LIN {X 0.073,Y -402.750,Z 613.612,A 0.000,B 0.000,C 90.000,E1 146.087} C_DIS
LIN {X 0.112,Y -403.409,Z 613.600,A 0.000,B 0.000,C 90.000,E1 143.989} C_DIS
LIN {X -0.051,Y -403.995,Z 613.590,A 0.000,B 0.000,C 90.000,E1 142.271} C_DIS
LIN {X -0.134,Y -404.710,Z 613.579,A 0.000,B 0.000,C 90.000,E1 140.194} C_DIS
LIN {X 0.098,Y -405.120,Z 613.571,A 0.000,B 0.000,C 90.000,E1 138.771} C_DIS
LIN {X -0.008,Y -405.586,Z 613.560,A 0.000,B 0.000,C 90.000,E1 136.701} C_DIS
LIN {X -0.089,Y -405.878,Z 613.552,A 0.000,B 0.000,C 90.000,E1 135.324} C_DIS
LIN {X -0.078,Y -406.430,Z 613.538,A 0.000,B 0.000,C 90.000,E1 132.894} C_DIS
LIN {X 0.152,Y -406.905,Z 613.527,A 0.000,B 0.000,C 90.000,E1 130.782} C_DIS
LIN {X -0.174,Y -407.650,Z 613.515,A 0.000,B 0.000,C 90.000,E1 128.749} C_DIS
LIN {X 0.026,Y -415.541,Z 613.500,A 0.000,B 0.000,C 90.000,E1 125.964} C_DIS
LIN {X -0.040,Y -419.640,Z 613.490,A 0.000,B 0.000,C 90.000,E1 124.246} C_DIS
LIN {X -0.079,Y -419.686,Z 613.490,A 0.000,B 0.000,C 90.000,E1 124.246} C_DIS
LIN {X 0.070,Y -424.345,Z 613.489,A 0.000,B 0.000,C 90.000,E1 123.913} C_DIS
LIN {X -0.100,Y -446.604,Z 613.482,A 0.000,B 0.000,C 90.000,E1 122.752} C_DIS
LIN {X 0.090,Y -454.993,Z 613.479,A 0.000,B 0.000,C 90.000,E1 122.291} C_DIS
LIN {X -0.061,Y -463.376,Z 613.477,A 0.000,B 0.000,C 90.000,E1 121.848} C_DIS
LIN {X 0.207,Y -474.847,Z 613.473,A 0.000,B 0.000,C 90.000,E1 121.131} C_DIS
LIN {X -0.221,Y -484.333,Z 613.470,A 0.000,B 0.000,C 90.000,E1 120.590} C_DIS
LIN {X -0.006,Y -489.087,Z 613.468,A 0.000,B 0.000,C 90.000,E1 120.256} C_DIS
LIN {X 0.293,Y -495.307,Z 613.466,A 0.000,B 0.000,C 90.000,E1 119.795} C_DIS
LIN {X -0.178,Y -502.690,Z 613.463,A 0.000,B 0.000,C 90.000,E1 119.333} C_DIS
LIN {X 0.224,Y -507.199,Z 613.461,A 0.000,B 0.000,C 90.000,E1 118.949} C_DIS
LIN {X -0.050,Y -514.629,Z 613.458,A 0.000,B 0.000,C 90.000,E1 118.409} C_DIS
LIN {X 0.031,Y -521.564,Z 613.455,A 0.000,B 0.000,C 90.000,E1 117.847} C_DIS
LIN {X -0.121,Y -528.772,Z 613.451,A 0.000,B 0.000,C 90.000,E1 117.257} C_DIS
LIN {X -0.178,Y -535.593,Z 613.448,A 0.000,B 0.000,C 90.000,E1 116.668} C_DIS
LIN {X -0.109,Y -540.696,Z 613.445,A 0.000,B 0.000,C 90.000,E1 116.181} C_DIS
LIN {X -0.107,Y -545.705,Z 613.443,A 0.000,B 0.000,C 90.000,E1 115.668} C_DIS
LIN {X 0.123,Y -550.229,Z 613.440,A 0.000,B 0.000,C 90.000,E1 115.155} C_DIS
LIN {X 0.197,Y -554.784,Z 613.437,A 0.000,B 0.000,C 90.000,E1 114.591} C_DIS
LIN {X 0.157,Y -559.646,Z 613.433,A 0.000,B 0.000,C 90.000,E1 113.898} C_DIS
LIN {X 0.159,Y -563.793,Z 613.429,A 0.000,B 0.000,C 90.000,E1 113.206} C_DIS
LIN {X 0.098,Y -568.224,Z 613.424,A 0.000,B 0.000,C 90.000,E1 112.386} C_DIS
LIN {X -0.137,Y -572.184,Z 613.420,A 0.000,B 0.000,C 90.000,E1 111.589} C_DIS
LIN {X -0.247,Y -575.292,Z 613.416,A 0.000,B 0.000,C 90.000,E1 110.918} C_DIS
LIN {X 0.130,Y -578.678,Z 613.412,A 0.000,B 0.000,C 90.000,E1 110.066} C_DIS
LIN {X -0.162,Y -582.700,Z 613.406,A 0.000,B 0.000,C 90.000,E1 109.014} C_DIS
LIN {X -0.112,Y -584.647,Z 613.403,A 0.000,B 0.000,C 90.000,E1 108.471} C_DIS
LIN {X 0.181,Y -587.212,Z 613.398,A 0.000,B 0.000,C 90.000,E1 107.638} C_DIS
LIN {X 0.193,Y -590.315,Z 613.392,A 0.000,B 0.000,C 90.000,E1 106.567} C_DIS
LIN {X -0.158,Y -593.106,Z 613.386,A 0.000,B 0.000,C 90.000,E1 105.536} C_DIS
LIN {X -0.083,Y -600.448,Z 613.372,A 0.000,B 0.000,C 90.000,E1 102.883} C_DIS
LIN {X 0.280,Y -604.239,Z 613.364,A 0.000,B 0.000,C 90.000,E1 101.535} C_DIS
LIN {X 0.267,Y -607.275,Z 613.358,A 0.000,B 0.000,C 90.000,E1 100.489} C_DIS
LIN {X 0.040,Y -610.915,Z 613.351,A 0.000,B 0.000,C 90.000,E1 99.208} C_DIS
LIN {X -0.225,Y -614.306,Z 613.344,A 0.000,B 0.000,C 90.000,E1 97.936} C_DIS
LIN {X -0.105,Y -616.905,Z 613.338,A 0.000,B 0.000,C 90.000,E1 96.891} C_DIS
LIN {X -0.031,Y -619.305,Z 613.333,A 0.000,B 0.000,C 90.000,E1 95.853} C_DIS
LIN {X -0.293,Y -620.884,Z 613.328,A 0.000,B 0.000,C 90.000,E1 95.106} C_DIS
LIN {X 0.152,Y -623.278,Z 613.321,A 0.000,B 0.000,C 90.000,E1 93.784} C_DIS
LIN {X 0.261,Y -624.948,Z 613.315,A 0.000,B 0.000,C 90.000,E1 92.751} C_DIS
LIN {X -0.235,Y -626.386,Z 613.310,A 0.000,B 0.000,C 90.000,E1 91.776} C_DIS
LIN {X -0.174,Y -627.104,Z 613.307,A 0.000,B 0.000,C 90.000,E1 91.260} C_DIS
LIN {X -0.031,Y -628.115,Z 613.301,A 0.000,B 0.000,C 90.000,E1 90.229} C_DIS
LIN {X -0.229,Y -628.671,Z 613.297,A 0.000,B 0.000,C 90.000,E1 89.484} C_DIS
LIN {X 0.206,Y -628.976,Z 613.293,A 0.000,B 0.000,C 90.000,E1 88.682} C_DIS
LIN {X -0.240,Y -629.148,Z 613.287,A 0.000,B 0.000,C 90.000,E1 87.707} C_DIS
LIN {X 0.191,Y -629.030,Z 613.283,A 0.000,B 0.000,C 90.000,E1 86.906} C_DIS
LIN {X 0.137,Y -628.580,Z 613.276,A 0.000,B 0.000,C 90.000,E1 85.641} C_DIS
LIN {X 0.082,Y -627.646,Z 613.269,A 0.000,B 0.000,C 90.000,E1 84.375} C_DIS
LIN {X 0.007,Y -626.487,Z 613.262,A 0.000,B 0.000,C 90.000,E1 83.109} C_DIS
LIN {X 0.287,Y -625.243,Z 613.256,A 0.000,B 0.000,C 90.000,E1 82.064} C_DIS
LIN {X -0.152,Y -623.664,Z 613.250,A 0.000,B 0.000,C 90.000,E1 81.084} C_DIS
LIN {X 0.263,Y -620.907,Z 613.242,A 0.000,B 0.000,C 90.000,E1 79.511} C_DIS
LIN {X -0.139,Y -618.827,Z 613.236,A 0.000,B 0.000,C 90.000,E1 78.522} C_DIS
LIN {X 0.158,Y -616.553,Z 613.230,A 0.000,B 0.000,C 90.000,E1 77.465} C_DIS
LIN {X -0.174,Y -614.146,Z 613.225,A 0.000,B 0.000,C 90.000,E1 76.464} C_DIS
LIN {X 0.054,Y -611.588,Z 613.219,A 0.000,B 0.000,C 90.000,E1 75.408} C_DIS
LIN {X -0.192,Y -608.825,Z 613.213,A 0.000,B 0.000,C 90.000,E1 74.393} C_DIS
LIN {X 0.113,Y -605.900,Z 613.207,A 0.000,B 0.000,C 90.000,E1 73.323} C_DIS
LIN {X 0.065,Y -603.504,Z 613.203,A 0.000,B 0.000,C 90.000,E1 72.543} C_DIS
LIN {X -0.009,Y -600.882,Z 613.199,A 0.000,B 0.000,C 90.000,E1 71.764} C_DIS
LIN {X -0.211,Y -596.826,Z 613.193,A 0.000,B 0.000,C 90.000,E1 70.732} C_DIS
LIN {X -0.156,Y -593.507,Z 613.188,A 0.000,B 0.000,C 90.000,E1 69.934} C_DIS
LIN {X 0.153,Y -589.410,Z 613.183,A 0.000,B 0.000,C 90.000,E1 68.975} C_DIS
LIN {X 0.151,Y -585.015,Z 613.178,A 0.000,B 0.000,C 90.000,E1 68.050} C_DIS
LIN {X -0.175,Y -581.595,Z 613.174,A 0.000,B 0.000,C 90.000,E1 67.411} C_DIS
LIN {X -0.287,Y -577.056,Z 613.170,A 0.000,B 0.000,C 90.000,E1 66.613} C_DIS
LIN {X -0.138,Y -572.989,Z 613.166,A 0.000,B 0.000,C 90.000,E1 65.921} C_DIS
LIN {X 0.057,Y -569.490,Z 613.163,A 0.000,B 0.000,C 90.000,E1 65.357} C_DIS
LIN {X 0.042,Y -563.363,Z 613.159,A 0.000,B 0.000,C 90.000,E1 64.537} C_DIS
LIN {X -0.244,Y -560.182,Z 613.156,A 0.000,B 0.000,C 90.000,E1 64.152} C_DIS
LIN {X -0.145,Y -555.580,Z 613.153,A 0.000,B 0.000,C 90.000,E1 63.589} C_DIS
LIN {X -0.107,Y -549.415,Z 613.150,A 0.000,B 0.000,C 90.000,E1 62.948} C_DIS
LIN {X -0.330,Y -544.196,Z 613.147,A 0.000,B 0.000,C 90.000,E1 62.487} C_DIS
LIN {X -0.241,Y -539.657,Z 613.145,A 0.000,B 0.000,C 90.000,E1 62.103} C_DIS
LIN {X -0.278,Y -534.953,Z 613.143,A 0.000,B 0.000,C 90.000,E1 61.769} C_DIS
LIN {X 0.296,Y -528.777,Z 613.141,A 0.000,B 0.000,C 90.000,E1 61.307} C_DIS
LIN {X 0.186,Y -521.819,Z 613.139,A 0.000,B 0.000,C 90.000,E1 60.923} C_DIS
LIN {X 0.085,Y -516.888,Z 613.137,A 0.000,B 0.000,C 90.000,E1 60.667} C_DIS
LIN {X 0.102,Y -504.926,Z 613.134,A 0.000,B 0.000,C 90.000,E1 60.078} C_DIS
LIN {X 0.043,Y -486.360,Z 613.129,A 0.000,B 0.000,C 90.000,E1 59.203} C_DIS
LIN {X -0.144,Y -467.737,Z 613.124,A 0.000,B 0.000,C 90.000,E1 58.329} C_DIS
LIN {X -0.119,Y -449.331,Z 613.119,A 0.000,B 0.000,C 90.000,E1 57.375} C_DIS
LIN {X -0.171,Y -445.106,Z 613.118,A 0.000,B 0.000,C 90.000,E1 57.168} C_DIS
LIN {X 0.161,Y -445.092,Z 613.117,A 0.000,B 0.000,C 90.000,E1 57.120} C_DIS
LIN {X 0.186,Y -443.839,Z 613.114,A 0.000,B 0.000,C 90.000,E1 56.421} C_DIS
LIN {X 0.198,Y -434.691,Z 613.092,A 0.000,B 0.000,C 90.000,E1 52.477} C_DIS
LIN {X -0.024,Y -431.565,Z 613.083,A 0.000,B 0.000,C 90.000,E1 50.848} C_DIS
LIN {X -0.023,Y -429.048,Z 613.077,A 0.000,B 0.000,C 90.000,E1 49.828} C_DIS
LIN {X 0.098,Y -430.066,Z 613.068,A 0.000,B 0.000,C 90.000,E1 48.162} C_DIS
LIN {X -0.021,Y -431.027,Z 613.057,A 0.000,B 0.000,C 90.000,E1 46.176} C_DIS
LIN {X -0.117,Y -431.999,Z 613.045,A 0.000,B 0.000,C 90.000,E1 44.190} C_DIS
LIN {X -0.131,Y -432.905,Z 613.036,A 0.000,B 0.000,C 90.000,E1 42.528} C_DIS
LIN {X -0.096,Y -433.765,Z 613.027,A 0.000,B 0.000,C 90.000,E1 40.862} C_DIS
LIN {X 0.224,Y -434.710,Z 613.016,A 0.000,B 0.000,C 90.000,E1 38.830} C_DIS
LIN {X -0.256,Y -435.438,Z 613.007,A 0.000,B 0.000,C 90.000,E1 37.237} C_DIS
LIN {X -0.037,Y -435.880,Z 612.999,A 0.000,B 0.000,C 90.000,E1 35.884} C_DIS
LIN {X -0.132,Y -436.474,Z 612.988,A 0.000,B 0.000,C 90.000,E1 33.913} C_DIS
LIN {X -0.074,Y -437.035,Z 612.976,A 0.000,B 0.000,C 90.000,E1 31.592} C_DIS
LIN {X -0.113,Y -437.511,Z 612.964,A 0.000,B 0.000,C 90.000,E1 29.617} C_DIS
LIN {X -0.167,Y -437.939,Z 612.955,A 0.000,B 0.000,C 90.000,E1 27.975} C_DIS
LIN {X -0.031,Y -438.353,Z 612.946,A 0.000,B 0.000,C 90.000,E1 26.309} C_DIS
LIN {X 0.110,Y -438.845,Z 612.937,A 0.000,B 0.000,C 90.000,E1 24.643} C_DIS
LIN {X -0.092,Y -439.468,Z 612.926,A 0.000,B 0.000,C 90.000,E1 22.695} C_DIS
LIN {X -0.055,Y -440.105,Z 612.917,A 0.000,B 0.000,C 90.000,E1 21.046} C_DIS
LIN {X 0.004,Y -440.804,Z 612.908,A 0.000,B 0.000,C 90.000,E1 19.396} C_DIS
LIN {X 0.039,Y -441.756,Z 612.895,A 0.000,B 0.000,C 90.000,E1 17.094} C_DIS
LIN {X -0.007,Y -442.725,Z 612.884,A 0.000,B 0.000,C 90.000,E1 15.134} C_DIS
LIN {X -0.136,Y -444.216,Z 612.870,A 0.000,B 0.000,C 90.000,E1 12.535} C_DIS
LIN {X 0.020,Y -446.045,Z 612.855,A 0.000,B 0.000,C 90.000,E1 9.905} C_DIS
LIN {X 0.155,Y -447.600,Z 612.844,A 0.000,B 0.000,C 90.000,E1 7.936} C_DIS
LIN {X 0.013,Y -449.613,Z 612.832,A 0.000,B 0.000,C 90.000,E1 5.682} C_DIS
LIN {X -0.166,Y -451.886,Z 612.819,A 0.000,B 0.000,C 90.000,E1 3.440} C_DIS
LIN {X 0.140,Y -454.456,Z 612.807,A 0.000,B 0.000,C 90.000,E1 1.146} C_DIS
LIN {X 0.189,Y -458.356,Z 612.790,A 0.000,B 0.000,C 90.000,E1 358.167} C_DIS
LIN {X -0.013,Y -462.209,Z 612.776,A 0.000,B 0.000,C 90.000,E1 355.641} C_DIS
LIN {X -0.054,Y -465.357,Z 612.765,A 0.000,B 0.000,C 90.000,E1 353.742} C_DIS
LIN {X 0.026,Y -468.480,Z 612.755,A 0.000,B 0.000,C 90.000,E1 351.837} C_DIS
LIN {X -0.046,Y -470.984,Z 612.746,A 0.000,B 0.000,C 90.000,E1 350.274} C_DIS
LIN {X 0.063,Y -475.111,Z 612.732,A 0.000,B 0.000,C 90.000,E1 347.757} C_DIS
LIN {X -0.049,Y -479.579,Z 612.718,A 0.000,B 0.000,C 90.000,E1 345.283} C_DIS
LIN {X 0.220,Y -484.136,Z 612.705,A 0.000,B 0.000,C 90.000,E1 342.779} C_DIS
LIN {X -0.052,Y -487.075,Z 612.696,A 0.000,B 0.000,C 90.000,E1 341.275} C_DIS
LIN {X -0.085,Y -490.625,Z 612.686,A 0.000,B 0.000,C 90.000,E1 339.444} C_DIS
LIN {X -0.086,Y -493.494,Z 612.677,A 0.000,B 0.000,C 90.000,E1 337.922} C_DIS
LIN {X -0.120,Y -496.091,Z 612.669,A 0.000,B 0.000,C 90.000,E1 336.410} C_DIS
LIN {X -0.092,Y -498.501,Z 612.661,A 0.000,B 0.000,C 90.000,E1 334.897} C_DIS
LIN {X -0.027,Y -500.785,Z 612.652,A 0.000,B 0.000,C 90.000,E1 333.384} C_DIS
LIN {X -0.148,Y -502.972,Z 612.644,A 0.000,B 0.000,C 90.000,E1 331.897} C_DIS
LIN {X 0.014,Y -505.164,Z 612.635,A 0.000,B 0.000,C 90.000,E1 330.383} C_DIS
LIN {X -0.159,Y -507.817,Z 612.626,A 0.000,B 0.000,C 90.000,E1 328.614} C_DIS
LIN {X -0.131,Y -514.434,Z 612.606,A 0.000,B 0.000,C 90.000,E1 325.055} C_DIS
LIN {X 0.056,Y -519.892,Z 612.593,A 0.000,B 0.000,C 90.000,E1 322.683} C_DIS
LIN {X 0.002,Y -520.753,Z 612.591,A 0.000,B 0.000,C 90.000,E1 322.396} C_DIS
LIN {X -0.102,Y -522.945,Z 612.588,A 0.000,B 0.000,C 90.000,E1 321.823} C_DIS
LIN {X -0.148,Y -524.574,Z 612.586,A 0.000,B 0.000,C 90.000,E1 321.537} C_DIS
LIN {X -0.189,Y -525.990,Z 612.585,A 0.000,B 0.000,C 90.000,E1 321.251} C_DIS
LIN {X 0.048,Y -527.317,Z 612.584,A 0.000,B 0.000,C 90.000,E1 321.045} C_DIS
LIN {X -0.096,Y -531.585,Z 612.581,A 0.000,B 0.000,C 90.000,E1 320.642} C_DIS
LIN {X 0.056,Y -534.164,Z 612.580,A 0.000,B 0.000,C 90.000,E1 320.356} C_DIS
LIN {X -0.202,Y -538.452,Z 612.578,A 0.000,B 0.000,C 90.000,E1 319.989} C_DIS
LIN {X 0.201,Y -546.399,Z 612.574,A 0.000,B 0.000,C 90.000,E1 319.299} C_DIS
LIN {X -0.149,Y -553.775,Z 612.571,A 0.000,B 0.000,C 90.000,E1 318.771} C_DIS
LIN {X -0.073,Y -565.332,Z 612.566,A 0.000,B 0.000,C 90.000,E1 317.838} C_DIS
LIN {X 0.137,Y -582.769,Z 612.558,A 0.000,B 0.000,C 90.000,E1 316.458} C_DIS
LIN {X -0.011,Y -592.437,Z 612.554,A 0.000,B 0.000,C 90.000,E1 315.688} C_DIS
LIN {X -0.204,Y -600.545,Z 612.550,A 0.000,B 0.000,C 90.000,E1 315.000} C_DIS
LIN {X -0.188,Y -605.824,Z 612.547,A 0.000,B 0.000,C 90.000,E1 314.514} C_DIS
LIN {X 0.077,Y -610.557,Z 612.545,A 0.000,B 0.000,C 90.000,E1 314.028} C_DIS
LIN {X -0.197,Y -616.178,Z 612.541,A 0.000,B 0.000,C 90.000,E1 313.461} C_DIS
LIN {X 0.289,Y -621.962,Z 612.538,A 0.000,B 0.000,C 90.000,E1 312.771} C_DIS
LIN {X -0.178,Y -629.472,Z 612.533,A 0.000,B 0.000,C 90.000,E1 311.919} C_DIS
LIN {X -0.168,Y -637.595,Z 612.527,A 0.000,B 0.000,C 90.000,E1 310.906} C_DIS
LIN {X 0.012,Y -645.331,Z 612.522,A 0.000,B 0.000,C 90.000,E1 309.886} C_DIS
LIN {X -0.148,Y -648.943,Z 612.519,A 0.000,B 0.000,C 90.000,E1 309.402} C_DIS
LIN {X -0.169,Y -652.357,Z 612.516,A 0.000,B 0.000,C 90.000,E1 308.910} C_DIS
LIN {X -0.245,Y -656.969,Z 612.512,A 0.000,B 0.000,C 90.000,E1 308.177} C_DIS
LIN {X -0.281,Y -661.142,Z 612.508,A 0.000,B 0.000,C 90.000,E1 307.443} C_DIS
LIN {X 0.204,Y -664.308,Z 612.505,A 0.000,B 0.000,C 90.000,E1 306.790} C_DIS
LIN {X -0.164,Y -667.776,Z 612.500,A 0.000,B 0.000,C 90.000,E1 306.091} C_DIS
LIN {X -0.111,Y -670.868,Z 612.496,A 0.000,B 0.000,C 90.000,E1 305.358} C_DIS
LIN {X 0.131,Y -673.678,Z 612.492,A 0.000,B 0.000,C 90.000,E1 304.612} C_DIS
LIN {X 0.011,Y -677.229,Z 612.487,A 0.000,B 0.000,C 90.000,E1 303.658} C_DIS
LIN {X 0.310,Y -680.526,Z 612.482,A 0.000,B 0.000,C 90.000,E1 302.673} C_DIS
LIN {X -0.110,Y -684.530,Z 612.475,A 0.000,B 0.000,C 90.000,E1 301.514} C_DIS
LIN {X -0.237,Y -688.382,Z 612.468,A 0.000,B 0.000,C 90.000,E1 300.335} C_DIS
LIN {X 0.045,Y -692.081,Z 612.462,A 0.000,B 0.000,C 90.000,E1 299.127} C_DIS
LIN {X 0.076,Y -694.898,Z 612.457,A 0.000,B 0.000,C 90.000,E1 298.180} C_DIS
LIN {X 0.224,Y -696.862,Z 612.453,A 0.000,B 0.000,C 90.000,E1 297.462} C_DIS
LIN {X -0.238,Y -698.624,Z 612.449,A 0.000,B 0.000,C 90.000,E1 296.796} C_DIS
LIN {X 0.025,Y -699.176,Z 612.448,A 0.000,B 0.000,C 90.000,E1 296.539} C_DIS
LIN {X -0.377,Y -699.690,Z 612.445,A 0.000,B 0.000,C 90.000,E1 296.104} C_DIS
LIN {X -0.108,Y -699.900,Z 612.444,A 0.000,B 0.000,C 90.000,E1 295.848} C_DIS
LIN {X 0.161,Y -699.634,Z 612.442,A 0.000,B 0.000,C 90.000,E1 295.591} C_DIS
LIN {X -0.230,Y -698.669,Z 612.440,A 0.000,B 0.000,C 90.000,E1 295.155} C_DIS
LIN {X 0.037,Y -697.532,Z 612.438,A 0.000,B 0.000,C 90.000,E1 294.899} C_DIS
LIN {X -0.363,Y -694.083,Z 612.436,A 0.000,B 0.000,C 90.000,E1 294.463} C_DIS
LIN {X -0.236,Y -692.863,Z 612.435,A 0.000,B 0.000,C 90.000,E1 294.335} C_DIS
LIN {X -0.111,Y -690.927,Z 612.435,A 0.000,B 0.000,C 90.000,E1 294.207} C_DIS
LIN {X -0.313,Y -683.658,Z 612.433,A 0.000,B 0.000,C 90.000,E1 293.898} C_DIS
LIN {X -0.239,Y -681.111,Z 612.432,A 0.000,B 0.000,C 90.000,E1 293.823} C_DIS
LIN {X 0.181,Y -677.794,Z 612.432,A 0.000,B 0.000,C 90.000,E1 293.718} C_DIS
LIN {X -0.189,Y -675.746,Z 612.432,A 0.000,B 0.000,C 90.000,E1 293.695} C_DIS
LIN {X -0.053,Y -668.987,Z 612.431,A 0.000,B 0.000,C 90.000,E1 293.590} C_DIS
LIN {X 0.379,Y -647.864,Z 612.429,A 0.000,B 0.000,C 90.000,E1 293.259} C_DIS
LIN {X -0.161,Y -638.051,Z 612.428,A 0.000,B 0.000,C 90.000,E1 293.131} C_DIS
LIN {X 0.139,Y -628.502,Z 612.427,A 0.000,B 0.000,C 90.000,E1 292.898} C_DIS
LIN {X -0.291,Y -621.940,Z 612.426,A 0.000,B 0.000,C 90.000,E1 292.770} C_DIS
LIN {X -0.213,Y -605.336,Z 612.424,A 0.000,B 0.000,C 90.000,E1 292.280} C_DIS
LIN {X 0.108,Y -581.030,Z 612.419,A 0.000,B 0.000,C 90.000,E1 291.482} C_DIS
LIN {X -0.168,Y -565.314,Z 612.417,A 0.000,B 0.000,C 90.000,E1 291.046} C_DIS
LIN {X -0.257,Y -559.795,Z 612.415,A 0.000,B 0.000,C 90.000,E1 290.791} C_DIS
LIN {X 0.095,Y -558.001,Z 612.414,A 0.000,B 0.000,C 90.000,E1 290.556} C_DIS
LIN {X 0.052,Y -557.961,Z 612.414,A 0.000,B 0.000,C 90.000,E1 290.556} C_DIS
LIN {X 0.091,Y -557.398,Z 612.413,A 0.000,B 0.000,C 90.000,E1 290.301} C_DIS
LIN {X 0.150,Y -557.281,Z 612.407,A 0.000,B 0.000,C 90.000,E1 289.322} C_DIS
LIN {X -0.093,Y -557.311,Z 612.401,A 0.000,B 0.000,C 90.000,E1 288.236} C_DIS
LIN {X 0.195,Y -557.177,Z 612.395,A 0.000,B 0.000,C 90.000,E1 287.094} C_DIS
LIN {X 0.068,Y -556.689,Z 612.387,A 0.000,B 0.000,C 90.000,E1 285.717} C_DIS
LIN {X 0.190,Y -556.176,Z 612.381,A 0.000,B 0.000,C 90.000,E1 284.592} C_DIS
LIN {X 0.021,Y -555.336,Z 612.372,A 0.000,B 0.000,C 90.000,E1 282.939} C_DIS
LIN {X 0.124,Y -554.619,Z 612.364,A 0.000,B 0.000,C 90.000,E1 281.535} C_DIS
LIN {X -0.182,Y -553.624,Z 612.353,A 0.000,B 0.000,C 90.000,E1 279.613} C_DIS
LIN {X -0.170,Y -552.772,Z 612.344,A 0.000,B 0.000,C 90.000,E1 277.936} C_DIS
LIN {X -0.174,Y -552.018,Z 612.335,A 0.000,B 0.000,C 90.000,E1 276.258} C_DIS
LIN {X -0.209,Y -551.322,Z 612.324,A 0.000,B 0.000,C 90.000,E1 274.302} C_DIS
LIN {X 0.192,Y -550.796,Z 612.315,A 0.000,B 0.000,C 90.000,E1 272.579} C_DIS
LIN {X 0.001,Y -550.375,Z 612.305,A 0.000,B 0.000,C 90.000,E1 270.917} C_DIS
LIN {X -0.264,Y -549.900,Z 612.297,A 0.000,B 0.000,C 90.000,E1 269.542} C_DIS
LIN {X -0.045,Y -549.494,Z 612.291,A 0.000,B 0.000,C 90.000,E1 268.396} C_DIS
LIN {X -0.240,Y -548.822,Z 612.282,A 0.000,B 0.000,C 90.000,E1 266.731} C_DIS
LIN {X 0.022,Y -548.164,Z 612.274,A 0.000,B 0.000,C 90.000,E1 265.298} C_DIS
LIN {X 0.235,Y -547.667,Z 612.269,A 0.000,B 0.000,C 90.000,E1 264.432} C_DIS
LIN {X -0.037,Y -546.717,Z 612.261,A 0.000,B 0.000,C 90.000,E1 263.053} C_DIS
LIN {X 0.256,Y -545.757,Z 612.255,A 0.000,B 0.000,C 90.000,E1 261.894} C_DIS
LIN {X 0.174,Y -543.811,Z 612.244,A 0.000,B 0.000,C 90.000,E1 259.926} C_DIS
LIN {X 0.233,Y -541.938,Z 612.233,A 0.000,B 0.000,C 90.000,E1 257.937} C_DIS
LIN {X 0.293,Y -540.376,Z 612.224,A 0.000,B 0.000,C 90.000,E1 256.228} C_DIS
LIN {X 0.187,Y -539.313,Z 612.217,A 0.000,B 0.000,C 90.000,E1 255.102} C_DIS
LIN {X -0.187,Y -537.471,Z 612.208,A 0.000,B 0.000,C 90.000,E1 253.433} C_DIS
LIN {X 0.068,Y -535.761,Z 612.198,A 0.000,B 0.000,C 90.000,E1 251.692} C_DIS
LIN {X -0.163,Y -534.849,Z 612.194,A 0.000,B 0.000,C 90.000,E1 250.859} C_DIS
LIN {X -0.033,Y -533.391,Z 612.187,A 0.000,B 0.000,C 90.000,E1 249.699} C_DIS
LIN {X 0.075,Y -531.579,Z 612.181,A 0.000,B 0.000,C 90.000,E1 248.539} C_DIS
LIN {X -0.138,Y -529.662,Z 612.174,A 0.000,B 0.000,C 90.000,E1 247.411} C_DIS
LIN {X 0.114,Y -527.559,Z 612.168,A 0.000,B 0.000,C 90.000,E1 246.230} C_DIS
LIN {X 0.159,Y -525.906,Z 612.163,A 0.000,B 0.000,C 90.000,E1 245.357} C_DIS
LIN {X 0.093,Y -523.479,Z 612.157,A 0.000,B 0.000,C 90.000,E1 244.204} C_DIS
LIN {X 0.082,Y -521.617,Z 612.152,A 0.000,B 0.000,C 90.000,E1 243.332} C_DIS
LIN {X 0.192,Y -519.031,Z 612.145,A 0.000,B 0.000,C 90.000,E1 242.153} C_DIS
LIN {X -0.067,Y -515.600,Z 612.137,A 0.000,B 0.000,C 90.000,E1 240.717} C_DIS
LIN {X -0.138,Y -510.750,Z 612.126,A 0.000,B 0.000,C 90.000,E1 238.663} C_DIS
LIN {X 0.073,Y -507.787,Z 612.119,A 0.000,B 0.000,C 90.000,E1 237.454} C_DIS
LIN {X 0.121,Y -503.823,Z 612.111,A 0.000,B 0.000,C 90.000,E1 235.960} C_DIS
LIN {X -0.040,Y -499.741,Z 612.103,A 0.000,B 0.000,C 90.000,E1 234.482} C_DIS
LIN {X 0.164,Y -492.615,Z 612.088,A 0.000,B 0.000,C 90.000,E1 231.743} C_DIS
LIN {X -0.130,Y -489.510,Z 612.081,A 0.000,B 0.000,C 90.000,E1 230.561} C_DIS
LIN {X 0.007,Y -484.105,Z 612.069,A 0.000,B 0.000,C 90.000,E1 228.405} C_DIS
LIN {X 0.022,Y -480.295,Z 612.060,A 0.000,B 0.000,C 90.000,E1 226.863} C_DIS
LIN {X 0.169,Y -474.919,Z 612.048,A 0.000,B 0.000,C 90.000,E1 224.676} C_DIS
LIN {X -0.152,Y -469.932,Z 612.036,A 0.000,B 0.000,C 90.000,E1 222.528} C_DIS
LIN {X 0.021,Y -465.706,Z 612.026,A 0.000,B 0.000,C 90.000,E1 220.620} C_DIS
LIN {X -0.206,Y -461.640,Z 612.015,A 0.000,B 0.000,C 90.000,E1 218.749} C_DIS
LIN {X 0.187,Y -457.715,Z 612.005,A 0.000,B 0.000,C 90.000,E1 216.790} C_DIS
LIN {X -0.052,Y -453.977,Z 611.994,A 0.000,B 0.000,C 90.000,E1 214.898} C_DIS
LIN {X -0.086,Y -450.972,Z 611.985,A 0.000,B 0.000,C 90.000,E1 213.293} C_DIS
LIN {X 0.100,Y -446.838,Z 611.972,A 0.000,B 0.000,C 90.000,E1 211.003} C_DIS
LIN {X -0.057,Y -442.807,Z 611.960,A 0.000,B 0.000,C 90.000,E1 208.743} C_DIS
LIN {X -0.235,Y -439.885,Z 611.951,A 0.000,B 0.000,C 90.000,E1 207.129} C_DIS
LIN {X -0.077,Y -436.992,Z 611.941,A 0.000,B 0.000,C 90.000,E1 205.463} C_DIS
LIN {X 0.057,Y -433.568,Z 611.930,A 0.000,B 0.000,C 90.000,E1 203.462} C_DIS
LIN {X -0.081,Y -429.697,Z 611.917,A 0.000,B 0.000,C 90.000,E1 201.153} C_DIS
LIN {X -0.046,Y -426.363,Z 611.906,A 0.000,B 0.000,C 90.000,E1 199.141} C_DIS
LIN {X -0.166,Y -422.730,Z 611.893,A 0.000,B 0.000,C 90.000,E1 196.804} C_DIS
LIN {X -0.148,Y -419.886,Z 611.882,A 0.000,B 0.000,C 90.000,E1 194.773} C_DIS
LIN {X -0.116,Y -417.892,Z 611.874,A 0.000,B 0.000,C 90.000,E1 193.411} C_DIS
LIN {X 0.015,Y -414.241,Z 611.861,A 0.000,B 0.000,C 90.000,E1 191.007} C_DIS
LIN {X -0.112,Y -411.019,Z 611.848,A 0.000,B 0.000,C 90.000,E1 188.624} C_DIS
LIN {X -0.027,Y -408.734,Z 611.838,A 0.000,B 0.000,C 90.000,E1 186.891} C_DIS
LIN {X -0.063,Y -406.082,Z 611.827,A 0.000,B 0.000,C 90.000,E1 184.821} C_DIS
LIN {X 0.119,Y -402.200,Z 611.807,A 0.000,B 0.000,C 90.000,E1 181.318} C_DIS
LIN {X 0.189,Y -399.814,Z 611.792,A 0.000,B 0.000,C 90.000,E1 178.511} C_DIS
LIN {X -0.169,Y -398.107,Z 611.776,A 0.000,B 0.000,C 90.000,E1 175.755} C_DIS
LIN {X -0.179,Y -397.092,Z 611.759,A 0.000,B 0.000,C 90.000,E1 172.591} C_DIS
LIN {X 0.005,Y -396.606,Z 611.743,A 0.000,B 0.000,C 90.000,E1 169.746} C_DIS
LIN {X -0.087,Y -396.597,Z 611.731,A 0.000,B 0.000,C 90.000,E1 167.645} C_DIS
LIN {X 0.025,Y -397.009,Z 611.716,A 0.000,B 0.000,C 90.000,E1 164.810} C_DIS
LIN {X -0.162,Y -397.489,Z 611.704,A 0.000,B 0.000,C 90.000,E1 162.725} C_DIS
LIN {X -0.098,Y -398.006,Z 611.692,A 0.000,B 0.000,C 90.000,E1 160.604} C_DIS
LIN {X -0.101,Y -398.587,Z 611.682,A 0.000,B 0.000,C 90.000,E1 158.847} C_DIS
LIN {X -0.106,Y -399.318,Z 611.671,A 0.000,B 0.000,C 90.000,E1 156.741} C_DIS
LIN {X -0.065,Y -400.275,Z 611.657,A 0.000,B 0.000,C 90.000,E1 154.280} C_DIS
LIN {X -0.006,Y -400.776,Z 611.649,A 0.000,B 0.000,C 90.000,E1 152.871} C_DIS
LIN {X 0.056,Y -401.335,Z 611.642,A 0.000,B 0.000,C 90.000,E1 151.463} C_DIS
LIN {X 0.190,Y -402.117,Z 611.628,A 0.000,B 0.000,C 90.000,E1 148.997} C_DIS
LIN {X 0.110,Y -402.732,Z 611.616,A 0.000,B 0.000,C 90.000,E1 146.914} C_DIS
LIN {X 0.041,Y -403.487,Z 611.603,A 0.000,B 0.000,C 90.000,E1 144.482} C_DIS
LIN {X 0.012,Y -404.158,Z 611.591,A 0.000,B 0.000,C 90.000,E1 142.396} C_DIS
LIN {X -0.184,Y -404.951,Z 611.578,A 0.000,B 0.000,C 90.000,E1 139.989} C_DIS
LIN {X -0.087,Y -405.262,Z 611.572,A 0.000,B 0.000,C 90.000,E1 138.933} C_DIS
LIN {X 0.086,Y -405.723,Z 611.560,A 0.000,B 0.000,C 90.000,E1 136.824} C_DIS
LIN {X 0.018,Y -406.008,Z 611.553,A 0.000,B 0.000,C 90.000,E1 135.445} C_DIS
LIN {X 0.041,Y -406.507,Z 611.539,A 0.000,B 0.000,C 90.000,E1 133.014} C_DIS
LIN {X -0.188,Y -407.039,Z 611.526,A 0.000,B 0.000,C 90.000,E1 130.620} C_DIS
LIN {X 0.142,Y -407.689,Z 611.515,A 0.000,B 0.000,C 90.000,E1 128.669} C_DIS
LIN {X 0.092,Y -415.124,Z 611.501,A 0.000,B 0.000,C 90.000,E1 126.091} C_DIS
LIN {X 0.024,Y -416.038,Z 611.499,A 0.000,B 0.000,C 90.000,E1 125.758} C_DIS
LIN {X -0.191,Y -420.329,Z 611.489,A 0.000,B 0.000,C 90.000,E1 123.992} C_DIS
LIN {X -0.230,Y -420.357,Z 611.489,A 0.000,B 0.000,C 90.000,E1 123.992} C_DIS
LIN {X 0.079,Y -423.950,Z 611.487,A 0.000,B 0.000,C 90.000,E1 123.706} C_DIS
LIN {X 0.094,Y -431.463,Z 611.485,A 0.000,B 0.000,C 90.000,E1 123.293} C_DIS
LIN {X -0.141,Y -452.062,Z 611.479,A 0.000,B 0.000,C 90.000,E1 122.260} C_DIS
LIN {X 0.123,Y -458.727,Z 611.477,A 0.000,B 0.000,C 90.000,E1 121.878} C_DIS
LIN {X -0.150,Y -465.286,Z 611.475,A 0.000,B 0.000,C 90.000,E1 121.544} C_DIS
LIN {X -0.017,Y -476.739,Z 611.471,A 0.000,B 0.000,C 90.000,E1 120.846} C_DIS
LIN {X 0.137,Y -481.487,Z 611.470,A 0.000,B 0.000,C 90.000,E1 120.541} C_DIS
LIN {X -0.005,Y -489.375,Z 611.467,A 0.000,B 0.000,C 90.000,E1 120.050} C_DIS
LIN {X -0.010,Y -498.896,Z 611.463,A 0.000,B 0.000,C 90.000,E1 119.411} C_DIS
LIN {X 0.058,Y -503.560,Z 611.462,A 0.000,B 0.000,C 90.000,E1 119.077} C_DIS
LIN {X 0.152,Y -515.545,Z 611.457,A 0.000,B 0.000,C 90.000,E1 118.153} C_DIS
LIN {X -0.245,Y -520.061,Z 611.455,A 0.000,B 0.000,C 90.000,E1 117.847} C_DIS
LIN {X -0.199,Y -530.187,Z 611.450,A 0.000,B 0.000,C 90.000,E1 117.001} C_DIS
LIN {X -0.006,Y -535.818,Z 611.447,A 0.000,B 0.000,C 90.000,E1 116.488} C_DIS
LIN {X 0.002,Y -539.978,Z 611.445,A 0.000,B 0.000,C 90.000,E1 116.104} C_DIS
LIN {X -0.188,Y -546.468,Z 611.441,A 0.000,B 0.000,C 90.000,E1 115.463} C_DIS
LIN {X 0.136,Y -549.085,Z 611.440,A 0.000,B 0.000,C 90.000,E1 115.155} C_DIS
LIN {X 0.200,Y -553.345,Z 611.437,A 0.000,B 0.000,C 90.000,E1 114.643} C_DIS
LIN {X 0.353,Y -555.277,Z 611.436,A 0.000,B 0.000,C 90.000,E1 114.387} C_DIS
LIN {X -0.319,Y -559.305,Z 611.433,A 0.000,B 0.000,C 90.000,E1 113.898} C_DIS
LIN {X 0.018,Y -563.406,Z 611.429,A 0.000,B 0.000,C 90.000,E1 113.206} C_DIS
LIN {X -0.046,Y -567.962,Z 611.424,A 0.000,B 0.000,C 90.000,E1 112.386} C_DIS
LIN {X 0.247,Y -572.032,Z 611.420,A 0.000,B 0.000,C 90.000,E1 111.535} C_DIS
LIN {X 0.140,Y -575.213,Z 611.416,A 0.000,B 0.000,C 90.000,E1 110.865} C_DIS
LIN {X -0.020,Y -578.685,Z 611.411,A 0.000,B 0.000,C 90.000,E1 110.066} C_DIS
LIN {X 0.239,Y -582.782,Z 611.406,A 0.000,B 0.000,C 90.000,E1 108.960} C_DIS
LIN {X 0.293,Y -584.751,Z 611.403,A 0.000,B 0.000,C 90.000,E1 108.417} C_DIS
LIN {X -0.196,Y -586.585,Z 611.400,A 0.000,B 0.000,C 90.000,E1 107.928} C_DIS
LIN {X 0.045,Y -590.577,Z 611.392,A 0.000,B 0.000,C 90.000,E1 106.567} C_DIS
LIN {X 0.269,Y -593.422,Z 611.386,A 0.000,B 0.000,C 90.000,E1 105.481} C_DIS
LIN {X -0.218,Y -600.826,Z 611.372,A 0.000,B 0.000,C 90.000,E1 102.883} C_DIS
LIN {X 0.152,Y -604.672,Z 611.364,A 0.000,B 0.000,C 90.000,E1 101.535} C_DIS
LIN {X 0.144,Y -607.746,Z 611.358,A 0.000,B 0.000,C 90.000,E1 100.489} C_DIS
LIN {X -0.075,Y -611.430,Z 611.351,A 0.000,B 0.000,C 90.000,E1 99.208} C_DIS
LIN {X 0.010,Y -614.216,Z 611.345,A 0.000,B 0.000,C 90.000,E1 98.163} C_DIS
LIN {X -0.204,Y -617.511,Z 611.338,A 0.000,B 0.000,C 90.000,E1 96.891} C_DIS
LIN {X -0.122,Y -619.963,Z 611.333,A 0.000,B 0.000,C 90.000,E1 95.853} C_DIS
LIN {X 0.241,Y -621.548,Z 611.328,A 0.000,B 0.000,C 90.000,E1 95.049} C_DIS
LIN {X -0.246,Y -623.534,Z 611.323,A 0.000,B 0.000,C 90.000,E1 94.069} C_DIS
LIN {X -0.138,Y -625.275,Z 611.317,A 0.000,B 0.000,C 90.000,E1 93.037} C_DIS
LIN {X -0.029,Y -626.791,Z 611.311,A 0.000,B 0.000,C 90.000,E1 92.007} C_DIS
LIN {X 0.126,Y -628.111,Z 611.306,A 0.000,B 0.000,C 90.000,E1 90.974} C_DIS
LIN {X 0.283,Y -629.073,Z 611.300,A 0.000,B 0.000,C 90.000,E1 89.943} C_DIS
LIN {X -0.177,Y -629.667,Z 611.294,A 0.000,B 0.000,C 90.000,E1 88.969} C_DIS
LIN {X 0.015,Y -629.872,Z 611.289,A 0.000,B 0.000,C 90.000,E1 87.936} C_DIS
LIN {X 0.184,Y -629.777,Z 611.283,A 0.000,B 0.000,C 90.000,E1 86.906} C_DIS
LIN {X -0.209,Y -629.364,Z 611.277,A 0.000,B 0.000,C 90.000,E1 85.927} C_DIS
LIN {X 0.262,Y -628.912,Z 611.273,A 0.000,B 0.000,C 90.000,E1 85.122} C_DIS
LIN {X -0.188,Y -628.086,Z 611.267,A 0.000,B 0.000,C 90.000,E1 84.147} C_DIS
LIN {X 0.327,Y -627.412,Z 611.263,A 0.000,B 0.000,C 90.000,E1 83.337} C_DIS
LIN {X 0.323,Y -625.832,Z 611.256,A 0.000,B 0.000,C 90.000,E1 82.064} C_DIS
LIN {X -0.109,Y -624.223,Z 611.250,A 0.000,B 0.000,C 90.000,E1 81.084} C_DIS
LIN {X -0.075,Y -621.901,Z 611.243,A 0.000,B 0.000,C 90.000,E1 79.803} C_DIS
LIN {X 0.145,Y -619.834,Z 611.238,A 0.000,B 0.000,C 90.000,E1 78.757} C_DIS
LIN {X -0.150,Y -617.590,Z 611.232,A 0.000,B 0.000,C 90.000,E1 77.757} C_DIS
LIN {X -0.102,Y -614.530,Z 611.225,A 0.000,B 0.000,C 90.000,E1 76.464} C_DIS
LIN {X -0.114,Y -611.243,Z 611.218,A 0.000,B 0.000,C 90.000,E1 75.172} C_DIS
LIN {X 0.221,Y -608.409,Z 611.212,A 0.000,B 0.000,C 90.000,E1 74.102} C_DIS
LIN {X -0.156,Y -604.542,Z 611.205,A 0.000,B 0.000,C 90.000,E1 72.834} C_DIS
LIN {X -0.213,Y -601.920,Z 611.200,A 0.000,B 0.000,C 90.000,E1 72.054} C_DIS
LIN {X -0.299,Y -598.913,Z 611.196,A 0.000,B 0.000,C 90.000,E1 71.275} C_DIS
LIN {X 0.340,Y -595.681,Z 611.191,A 0.000,B 0.000,C 90.000,E1 70.423} C_DIS
LIN {X 0.176,Y -592.227,Z 611.187,A 0.000,B 0.000,C 90.000,E1 69.645} C_DIS
LIN {X 0.181,Y -588.600,Z 611.183,A 0.000,B 0.000,C 90.000,E1 68.847} C_DIS
LIN {X 0.139,Y -584.663,Z 611.178,A 0.000,B 0.000,C 90.000,E1 68.050} C_DIS
LIN {X -0.190,Y -581.169,Z 611.174,A 0.000,B 0.000,C 90.000,E1 67.411} C_DIS
LIN {X -0.091,Y -577.401,Z 611.171,A 0.000,B 0.000,C 90.000,E1 66.741} C_DIS
LIN {X 0.267,Y -573.375,Z 611.167,A 0.000,B 0.000,C 90.000,E1 66.049} C_DIS
LIN {X -0.138,Y -568.851,Z 611.163,A 0.000,B 0.000,C 90.000,E1 65.409} C_DIS
LIN {X 0.073,Y -563.753,Z 611.160,A 0.000,B 0.000,C 90.000,E1 64.717} C_DIS
LIN {X 0.036,Y -559.689,Z 611.157,A 0.000,B 0.000,C 90.000,E1 64.204} C_DIS
LIN {X 0.239,Y -555.056,Z 611.154,A 0.000,B 0.000,C 90.000,E1 63.640} C_DIS
LIN {X -0.035,Y -549.799,Z 611.151,A 0.000,B 0.000,C 90.000,E1 63.127} C_DIS
LIN {X 0.043,Y -544.266,Z 611.148,A 0.000,B 0.000,C 90.000,E1 62.615} C_DIS
LIN {X 0.242,Y -539.820,Z 611.146,A 0.000,B 0.000,C 90.000,E1 62.231} C_DIS
LIN {X -0.133,Y -533.320,Z 611.143,A 0.000,B 0.000,C 90.000,E1 61.820} C_DIS
LIN {X -0.151,Y -528.347,Z 611.142,A 0.000,B 0.000,C 90.000,E1 61.513} C_DIS
LIN {X -0.222,Y -519.936,Z 611.139,A 0.000,B 0.000,C 90.000,E1 61.051} C_DIS
LIN {X -0.318,Y -514.795,Z 611.138,A 0.000,B 0.000,C 90.000,E1 60.795} C_DIS
LIN {X 0.059,Y -504.455,Z 611.135,A 0.000,B 0.000,C 90.000,E1 60.255} C_DIS
LIN {X -0.021,Y -487.414,Z 611.130,A 0.000,B 0.000,C 90.000,E1 59.459} C_DIS
LIN {X -0.115,Y -472.099,Z 611.126,A 0.000,B 0.000,C 90.000,E1 58.742} C_DIS
LIN {X 0.001,Y -448.664,Z 611.120,A 0.000,B 0.000,C 90.000,E1 57.533} C_DIS
LIN {X -0.019,Y -445.557,Z 611.119,A 0.000,B 0.000,C 90.000,E1 57.375} C_DIS
LIN {X -0.062,Y -445.507,Z 611.119,A 0.000,B 0.000,C 90.000,E1 57.375} C_DIS
LIN {X 0.036,Y -443.667,Z 611.113,A 0.000,B 0.000,C 90.000,E1 56.373} C_DIS
LIN {X 0.026,Y -434.554,Z 611.091,A 0.000,B 0.000,C 90.000,E1 52.431} C_DIS
LIN {X -0.206,Y -431.424,Z 611.082,A 0.000,B 0.000,C 90.000,E1 50.803} C_DIS
LIN {X -0.030,Y -429.479,Z 611.078,A 0.000,B 0.000,C 90.000,E1 49.989} C_DIS
LIN {X -0.049,Y -430.456,Z 611.069,A 0.000,B 0.000,C 90.000,E1 48.447} C_DIS
LIN {X -0.068,Y -431.299,Z 611.060,A 0.000,B 0.000,C 90.000,E1 46.782} C_DIS
LIN {X 0.204,Y -432.153,Z 611.051,A 0.000,B 0.000,C 90.000,E1 45.081} C_DIS
LIN {X 0.073,Y -433.469,Z 611.038,A 0.000,B 0.000,C 90.000,E1 42.771} C_DIS
LIN {X -0.206,Y -434.326,Z 611.029,A 0.000,B 0.000,C 90.000,E1 41.148} C_DIS
LIN {X -0.145,Y -435.135,Z 611.019,A 0.000,B 0.000,C 90.000,E1 39.483} C_DIS
LIN {X -0.009,Y -435.893,Z 611.010,A 0.000,B 0.000,C 90.000,E1 37.810} C_DIS
LIN {X -0.134,Y -436.383,Z 611.003,A 0.000,B 0.000,C 90.000,E1 36.503} C_DIS
LIN {X 0.139,Y -436.976,Z 610.992,A 0.000,B 0.000,C 90.000,E1 34.485} C_DIS
LIN {X 0.159,Y -437.348,Z 610.983,A 0.000,B 0.000,C 90.000,E1 32.832} C_DIS
LIN {X -0.019,Y -437.768,Z 610.972,A 0.000,B 0.000,C 90.000,E1 30.875} C_DIS
LIN {X 0.149,Y -438.142,Z 610.962,A 0.000,B 0.000,C 90.000,E1 29.205} C_DIS
LIN {X -0.106,Y -438.568,Z 610.953,A 0.000,B 0.000,C 90.000,E1 27.590} C_DIS
LIN {X 0.209,Y -438.863,Z 610.946,A 0.000,B 0.000,C 90.000,E1 26.232} C_DIS
LIN {X 0.172,Y -439.334,Z 610.937,A 0.000,B 0.000,C 90.000,E1 24.591} C_DIS
LIN {X 0.141,Y -439.838,Z 610.928,A 0.000,B 0.000,C 90.000,E1 22.950} C_DIS
LIN {X -0.061,Y -440.410,Z 610.919,A 0.000,B 0.000,C 90.000,E1 21.334} C_DIS
LIN {X 0.109,Y -441.190,Z 610.908,A 0.000,B 0.000,C 90.000,E1 19.341} C_DIS
LIN {X 0.160,Y -442.119,Z 610.895,A 0.000,B 0.000,C 90.000,E1 17.040} C_DIS
LIN {X 0.128,Y -443.042,Z 610.884,A 0.000,B 0.000,C 90.000,E1 15.079} C_DIS
LIN {X -0.153,Y -444.323,Z 610.871,A 0.000,B 0.000,C 90.000,E1 12.827} C_DIS
LIN {X 0.006,Y -446.083,Z 610.857,A 0.000,B 0.000,C 90.000,E1 10.197} C_DIS
LIN {X 0.208,Y -447.610,Z 610.846,A 0.000,B 0.000,C 90.000,E1 8.219} C_DIS
LIN {X 0.198,Y -449.838,Z 610.831,A 0.000,B 0.000,C 90.000,E1 5.625} C_DIS
LIN {X 0.027,Y -452.113,Z 610.819,A 0.000,B 0.000,C 90.000,E1 3.383} C_DIS
LIN {X -0.115,Y -454.656,Z 610.806,A 0.000,B 0.000,C 90.000,E1 1.146} C_DIS
LIN {X 0.191,Y -458.516,Z 610.790,A 0.000,B 0.000,C 90.000,E1 358.167} C_DIS
LIN {X -0.006,Y -462.334,Z 610.776,A 0.000,B 0.000,C 90.000,E1 355.641} C_DIS
LIN {X -0.043,Y -465.460,Z 610.765,A 0.000,B 0.000,C 90.000,E1 353.742} C_DIS
LIN {X -0.232,Y -468.045,Z 610.756,A 0.000,B 0.000,C 90.000,E1 352.186} C_DIS
LIN {X 0.149,Y -470.560,Z 610.748,A 0.000,B 0.000,C 90.000,E1 350.566} C_DIS
LIN {X 0.079,Y -475.175,Z 610.732,A 0.000,B 0.000,C 90.000,E1 347.757} C_DIS
LIN {X -0.031,Y -479.610,Z 610.718,A 0.000,B 0.000,C 90.000,E1 345.283} C_DIS
LIN {X -0.073,Y -482.999,Z 610.708,A 0.000,B 0.000,C 90.000,E1 343.433} C_DIS
LIN {X 0.095,Y -485.324,Z 610.701,A 0.000,B 0.000,C 90.000,E1 342.181} C_DIS
LIN {X -0.017,Y -487.690,Z 610.694,A 0.000,B 0.000,C 90.000,E1 340.967} C_DIS
LIN {X -0.064,Y -490.656,Z 610.686,A 0.000,B 0.000,C 90.000,E1 339.444} C_DIS
LIN {X -0.065,Y -493.552,Z 610.677,A 0.000,B 0.000,C 90.000,E1 337.922} C_DIS
LIN {X -0.097,Y -496.119,Z 610.669,A 0.000,B 0.000,C 90.000,E1 336.410} C_DIS
LIN {X -0.069,Y -498.559,Z 610.661,A 0.000,B 0.000,C 90.000,E1 334.897} C_DIS
LIN {X -0.001,Y -500.845,Z 610.652,A 0.000,B 0.000,C 90.000,E1 333.384} C_DIS
LIN {X -0.036,Y -502.132,Z 610.647,A 0.000,B 0.000,C 90.000,E1 332.487} C_DIS
LIN {X 0.108,Y -504.363,Z 610.639,A 0.000,B 0.000,C 90.000,E1 330.973} C_DIS
LIN {X -0.076,Y -506.963,Z 610.629,A 0.000,B 0.000,C 90.000,E1 329.203} C_DIS
LIN {X -0.103,Y -514.382,Z 610.606,A 0.000,B 0.000,C 90.000,E1 325.055} C_DIS
LIN {X 0.027,Y -520.330,Z 610.591,A 0.000,B 0.000,C 90.000,E1 322.396} C_DIS
LIN {X 0.275,Y -522.260,Z 610.588,A 0.000,B 0.000,C 90.000,E1 321.823} C_DIS
LIN {X 0.227,Y -523.121,Z 610.586,A 0.000,B 0.000,C 90.000,E1 321.537} C_DIS
LIN {X -0.086,Y -524.628,Z 610.585,A 0.000,B 0.000,C 90.000,E1 321.251} C_DIS
LIN {X 0.130,Y -525.499,Z 610.583,A 0.000,B 0.000,C 90.000,E1 321.009} C_DIS
LIN {X 0.019,Y -527.107,Z 610.582,A 0.000,B 0.000,C 90.000,E1 320.803} C_DIS
LIN {X 0.163,Y -530.922,Z 610.580,A 0.000,B 0.000,C 90.000,E1 320.356} C_DIS
LIN {X -0.144,Y -535.803,Z 610.577,A 0.000,B 0.000,C 90.000,E1 319.908} C_DIS
LIN {X 0.080,Y -542.605,Z 610.574,A 0.000,B 0.000,C 90.000,E1 319.299} C_DIS
LIN {X 0.190,Y -547.061,Z 610.572,A 0.000,B 0.000,C 90.000,E1 318.933} C_DIS
LIN {X 0.027,Y -551.622,Z 610.570,A 0.000,B 0.000,C 90.000,E1 318.609} C_DIS
LIN {X 0.182,Y -564.608,Z 610.564,A 0.000,B 0.000,C 90.000,E1 317.553} C_DIS
LIN {X 0.044,Y -582.117,Z 610.557,A 0.000,B 0.000,C 90.000,E1 316.215} C_DIS
LIN {X -0.136,Y -590.512,Z 610.553,A 0.000,B 0.000,C 90.000,E1 315.567} C_DIS
LIN {X 0.103,Y -595.939,Z 610.551,A 0.000,B 0.000,C 90.000,E1 315.081} C_DIS
LIN {X 0.260,Y -604.109,Z 610.547,A 0.000,B 0.000,C 90.000,E1 314.352} C_DIS
LIN {X 0.126,Y -610.149,Z 610.543,A 0.000,B 0.000,C 90.000,E1 313.785} C_DIS
LIN {X 0.017,Y -613.815,Z 610.541,A 0.000,B 0.000,C 90.000,E1 313.419} C_DIS
LIN {X -0.370,Y -620.830,Z 610.537,A 0.000,B 0.000,C 90.000,E1 312.690} C_DIS
LIN {X 0.089,Y -628.401,Z 610.532,A 0.000,B 0.000,C 90.000,E1 311.757} C_DIS
LIN {X 0.078,Y -636.621,Z 610.526,A 0.000,B 0.000,C 90.000,E1 310.744} C_DIS
LIN {X 0.246,Y -644.459,Z 610.521,A 0.000,B 0.000,C 90.000,E1 309.725} C_DIS
LIN {X 0.087,Y -649.012,Z 610.517,A 0.000,B 0.000,C 90.000,E1 309.116} C_DIS
LIN {X 0.025,Y -651.609,Z 610.515,A 0.000,B 0.000,C 90.000,E1 308.749} C_DIS
LIN {X 0.429,Y -655.525,Z 610.512,A 0.000,B 0.000,C 90.000,E1 308.096} C_DIS
LIN {X -0.054,Y -659.143,Z 610.508,A 0.000,B 0.000,C 90.000,E1 307.523} C_DIS
LIN {X -0.025,Y -661.819,Z 610.506,A 0.000,B 0.000,C 90.000,E1 307.030} C_DIS
LIN {X 0.024,Y -664.310,Z 610.503,A 0.000,B 0.000,C 90.000,E1 306.537} C_DIS
LIN {X -0.449,Y -666.672,Z 610.500,A 0.000,B 0.000,C 90.000,E1 306.091} C_DIS
LIN {X 0.138,Y -669.821,Z 610.496,A 0.000,B 0.000,C 90.000,E1 305.311} C_DIS
LIN {X -0.178,Y -672.693,Z 610.492,A 0.000,B 0.000,C 90.000,E1 304.612} C_DIS
LIN {X 0.064,Y -676.305,Z 610.487,A 0.000,B 0.000,C 90.000,E1 303.627} C_DIS
LIN {X 0.153,Y -680.475,Z 610.480,A 0.000,B 0.000,C 90.000,E1 302.418} C_DIS
LIN {X -0.059,Y -685.276,Z 610.472,A 0.000,B 0.000,C 90.000,E1 301.003} C_DIS
LIN {X 0.181,Y -689.113,Z 610.466,A 0.000,B 0.000,C 90.000,E1 299.795} C_DIS
LIN {X 0.135,Y -692.853,Z 610.459,A 0.000,B 0.000,C 90.000,E1 298.615} C_DIS
LIN {X -0.108,Y -695.589,Z 610.454,A 0.000,B 0.000,C 90.000,E1 297.692} C_DIS
LIN {X -0.282,Y -697.461,Z 610.450,A 0.000,B 0.000,C 90.000,E1 297.001} C_DIS
LIN {X 0.241,Y -698.561,Z 610.447,A 0.000,B 0.000,C 90.000,E1 296.488} C_DIS
LIN {X -0.162,Y -699.051,Z 610.445,A 0.000,B 0.000,C 90.000,E1 296.052} C_DIS
LIN {X 0.106,Y -699.234,Z 610.443,A 0.000,B 0.000,C 90.000,E1 295.796} C_DIS
LIN {X 0.276,Y -697.899,Z 610.440,A 0.000,B 0.000,C 90.000,E1 295.079} C_DIS
LIN {X 0.113,Y -697.340,Z 610.439,A 0.000,B 0.000,C 90.000,E1 294.975} C_DIS
LIN {X 0.281,Y -693.156,Z 610.436,A 0.000,B 0.000,C 90.000,E1 294.387} C_DIS
LIN {X 0.120,Y -691.734,Z 610.435,A 0.000,B 0.000,C 90.000,E1 294.283} C_DIS
LIN {X -0.141,Y -686.078,Z 610.433,A 0.000,B 0.000,C 90.000,E1 294.027} C_DIS
LIN {X 0.392,Y -682.259,Z 610.433,A 0.000,B 0.000,C 90.000,E1 293.823} C_DIS
LIN {X -0.187,Y -675.073,Z 610.432,A 0.000,B 0.000,C 90.000,E1 293.695} C_DIS
LIN {X -0.045,Y -649.733,Z 610.430,A 0.000,B 0.000,C 90.000,E1 293.334} C_DIS
LIN {X 0.045,Y -639.779,Z 610.429,A 0.000,B 0.000,C 90.000,E1 293.153} C_DIS
LIN {X -0.016,Y -629.704,Z 610.428,A 0.000,B 0.000,C 90.000,E1 292.950} C_DIS
LIN {X -0.082,Y -620.309,Z 610.426,A 0.000,B 0.000,C 90.000,E1 292.717} C_DIS
LIN {X 0.001,Y -603.287,Z 610.423,A 0.000,B 0.000,C 90.000,E1 292.206} C_DIS
LIN {X 0.105,Y -582.395,Z 610.420,A 0.000,B 0.000,C 90.000,E1 291.535} C_DIS
LIN {X -0.082,Y -574.951,Z 610.419,A 0.000,B 0.000,C 90.000,E1 291.334} C_DIS
LIN {X -0.258,Y -564.923,Z 610.417,A 0.000,B 0.000,C 90.000,E1 291.046} C_DIS
LIN {X 0.167,Y -559.633,Z 610.415,A 0.000,B 0.000,C 90.000,E1 290.737} C_DIS
LIN {X -0.157,Y -558.198,Z 610.414,A 0.000,B 0.000,C 90.000,E1 290.610} C_DIS
LIN {X -0.199,Y -558.187,Z 610.414,A 0.000,B 0.000,C 90.000,E1 290.610} C_DIS
LIN {X 0.011,Y -557.639,Z 610.413,A 0.000,B 0.000,C 90.000,E1 290.355} C_DIS
LIN {X -0.109,Y -557.395,Z 610.410,A 0.000,B 0.000,C 90.000,E1 289.812} C_DIS
LIN {X 0.179,Y -557.511,Z 610.404,A 0.000,B 0.000,C 90.000,E1 288.671} C_DIS
LIN {X 0.236,Y -557.356,Z 610.396,A 0.000,B 0.000,C 90.000,E1 287.275} C_DIS
LIN {X 0.115,Y -556.917,Z 610.388,A 0.000,B 0.000,C 90.000,E1 285.898} C_DIS
LIN {X 0.241,Y -556.407,Z 610.382,A 0.000,B 0.000,C 90.000,E1 284.773} C_DIS
LIN {X 0.081,Y -555.577,Z 610.373,A 0.000,B 0.000,C 90.000,E1 283.119} C_DIS
LIN {X 0.193,Y -554.865,Z 610.365,A 0.000,B 0.000,C 90.000,E1 281.715} C_DIS
LIN {X -0.100,Y -553.865,Z 610.354,A 0.000,B 0.000,C 90.000,E1 279.792} C_DIS
LIN {X 0.120,Y -552.863,Z 610.344,A 0.000,B 0.000,C 90.000,E1 277.814} C_DIS
LIN {X -0.002,Y -552.205,Z 610.336,A 0.000,B 0.000,C 90.000,E1 276.429} C_DIS
LIN {X -0.039,Y -551.501,Z 610.325,A 0.000,B 0.000,C 90.000,E1 274.473} C_DIS
LIN {X -0.131,Y -550.868,Z 610.314,A 0.000,B 0.000,C 90.000,E1 272.522} C_DIS
LIN {X 0.174,Y -550.535,Z 610.306,A 0.000,B 0.000,C 90.000,E1 271.088} C_DIS
LIN {X -0.089,Y -550.077,Z 610.298,A 0.000,B 0.000,C 90.000,E1 269.714} C_DIS
LIN {X 0.186,Y -549.576,Z 610.291,A 0.000,B 0.000,C 90.000,E1 268.282} C_DIS
LIN {X -0.007,Y -548.905,Z 610.281,A 0.000,B 0.000,C 90.000,E1 266.617} C_DIS
LIN {X -0.293,Y -548.238,Z 610.273,A 0.000,B 0.000,C 90.000,E1 265.241} C_DIS
LIN {X -0.045,Y -547.544,Z 610.267,A 0.000,B 0.000,C 90.000,E1 264.090} C_DIS
LIN {X 0.258,Y -546.778,Z 610.261,A 0.000,B 0.000,C 90.000,E1 262.932} C_DIS
LIN {X -0.058,Y -545.813,Z 610.255,A 0.000,B 0.000,C 90.000,E1 261.837} C_DIS
LIN {X -0.135,Y -544.195,Z 610.245,A 0.000,B 0.000,C 90.000,E1 260.151} C_DIS
LIN {X -0.082,Y -542.013,Z 610.233,A 0.000,B 0.000,C 90.000,E1 257.881} C_DIS
LIN {X -0.022,Y -540.447,Z 610.223,A 0.000,B 0.000,C 90.000,E1 256.172} C_DIS
LIN {X -0.130,Y -539.334,Z 610.217,A 0.000,B 0.000,C 90.000,E1 255.046} C_DIS
LIN {X 0.008,Y -537.508,Z 610.207,A 0.000,B 0.000,C 90.000,E1 253.323} C_DIS
LIN {X -0.253,Y -535.815,Z 610.198,A 0.000,B 0.000,C 90.000,E1 251.638} C_DIS
LIN {X 0.195,Y -534.873,Z 610.193,A 0.000,B 0.000,C 90.000,E1 250.732} C_DIS
LIN {X -0.172,Y -533.372,Z 610.187,A 0.000,B 0.000,C 90.000,E1 249.625} C_DIS
LIN {X 0.137,Y -531.079,Z 610.179,A 0.000,B 0.000,C 90.000,E1 248.156} C_DIS
LIN {X -0.283,Y -529.057,Z 610.172,A 0.000,B 0.000,C 90.000,E1 247.050} C_DIS
LIN {X -0.046,Y -526.936,Z 610.166,A 0.000,B 0.000,C 90.000,E1 245.869} C_DIS
LIN {X -0.102,Y -524.581,Z 610.160,A 0.000,B 0.000,C 90.000,E1 244.717} C_DIS
LIN {X -0.032,Y -521.478,Z 610.151,A 0.000,B 0.000,C 90.000,E1 243.256} C_DIS
LIN {X -0.162,Y -518.852,Z 610.145,A 0.000,B 0.000,C 90.000,E1 242.103} C_DIS
LIN {X 0.274,Y -515.395,Z 610.137,A 0.000,B 0.000,C 90.000,E1 240.589} C_DIS
LIN {X 0.192,Y -510.529,Z 610.125,A 0.000,B 0.000,C 90.000,E1 238.535} C_DIS
LIN {X 0.067,Y -508.351,Z 610.120,A 0.000,B 0.000,C 90.000,E1 237.661} C_DIS
LIN {X 0.125,Y -504.364,Z 610.112,A 0.000,B 0.000,C 90.000,E1 236.167} C_DIS
LIN {X -0.026,Y -500.270,Z 610.104,A 0.000,B 0.000,C 90.000,E1 234.689} C_DIS
LIN {X 0.177,Y -494.585,Z 610.092,A 0.000,B 0.000,C 90.000,E1 232.557} C_DIS
LIN {X -0.242,Y -490.782,Z 610.084,A 0.000,B 0.000,C 90.000,E1 231.090} C_DIS
LIN {X 0.072,Y -484.557,Z 610.070,A 0.000,B 0.000,C 90.000,E1 228.609} C_DIS
LIN {X -0.099,Y -479.964,Z 610.060,A 0.000,B 0.000,C 90.000,E1 226.782} C_DIS
LIN {X -0.066,Y -475.352,Z 610.050,A 0.000,B 0.000,C 90.000,E1 224.919} C_DIS
LIN {X 0.294,Y -470.345,Z 610.037,A 0.000,B 0.000,C 90.000,E1 222.690} C_DIS
LIN {X -0.121,Y -465.392,Z 610.025,A 0.000,B 0.000,C 90.000,E1 220.539} C_DIS
LIN {X 0.038,Y -460.692,Z 610.013,A 0.000,B 0.000,C 90.000,E1 218.302} C_DIS
LIN {X 0.132,Y -456.772,Z 610.002,A 0.000,B 0.000,C 90.000,E1 216.377} C_DIS
LIN {X 0.058,Y -454.311,Z 609.995,A 0.000,B 0.000,C 90.000,E1 215.105} C_DIS
LIN {X 0.029,Y -451.265,Z 609.986,A 0.000,B 0.000,C 90.000,E1 213.499} C_DIS
LIN {X -0.159,Y -447.132,Z 609.974,A 0.000,B 0.000,C 90.000,E1 211.258} C_DIS
LIN {X -0.042,Y -444.206,Z 609.965,A 0.000,B 0.000,C 90.000,E1 209.617} C_DIS
LIN {X 0.068,Y -440.790,Z 609.954,A 0.000,B 0.000,C 90.000,E1 207.641} C_DIS
LIN {X 0.077,Y -437.287,Z 609.943,A 0.000,B 0.000,C 90.000,E1 205.668} C_DIS
LIN {X -0.001,Y -434.424,Z 609.934,A 0.000,B 0.000,C 90.000,E1 204.027} C_DIS
LIN {X 0.075,Y -431.061,Z 609.922,A 0.000,B 0.000,C 90.000,E1 202.025} C_DIS
LIN {X -0.059,Y -428.337,Z 609.913,A 0.000,B 0.000,C 90.000,E1 200.375} C_DIS
LIN {X 0.147,Y -424.548,Z 609.900,A 0.000,B 0.000,C 90.000,E1 198.000} C_DIS
LIN {X 0.039,Y -420.661,Z 609.885,A 0.000,B 0.000,C 90.000,E1 195.315} C_DIS
LIN {X -0.159,Y -418.226,Z 609.876,A 0.000,B 0.000,C 90.000,E1 193.647} C_DIS
LIN {X -0.064,Y -415.053,Z 609.864,A 0.000,B 0.000,C 90.000,E1 191.591} C_DIS
LIN {X -0.129,Y -411.352,Z 609.849,A 0.000,B 0.000,C 90.000,E1 188.859} C_DIS
LIN {X -0.033,Y -409.091,Z 609.840,A 0.000,B 0.000,C 90.000,E1 187.125} C_DIS
LIN {X -0.010,Y -405.981,Z 609.826,A 0.000,B 0.000,C 90.000,E1 184.702} C_DIS
LIN {X 0.135,Y -402.130,Z 609.807,A 0.000,B 0.000,C 90.000,E1 181.203} C_DIS
LIN {X -0.195,Y -399.797,Z 609.791,A 0.000,B 0.000,C 90.000,E1 178.453} C_DIS
LIN {X 0.180,Y -397.981,Z 609.774,A 0.000,B 0.000,C 90.000,E1 175.241} C_DIS
LIN {X -0.117,Y -397.147,Z 609.758,A 0.000,B 0.000,C 90.000,E1 172.470} C_DIS
LIN {X 0.038,Y -396.734,Z 609.744,A 0.000,B 0.000,C 90.000,E1 169.982} C_DIS
LIN {X -0.053,Y -396.692,Z 609.733,A 0.000,B 0.000,C 90.000,E1 167.881} C_DIS
LIN {X 0.022,Y -397.146,Z 609.715,A 0.000,B 0.000,C 90.000,E1 164.700} C_DIS
LIN {X -0.124,Y -397.557,Z 609.705,A 0.000,B 0.000,C 90.000,E1 162.960} C_DIS
LIN {X -0.185,Y -398.097,Z 609.694,A 0.000,B 0.000,C 90.000,E1 160.859} C_DIS
LIN {X 0.024,Y -398.766,Z 609.682,A 0.000,B 0.000,C 90.000,E1 158.720} C_DIS
LIN {X -0.045,Y -399.410,Z 609.672,A 0.000,B 0.000,C 90.000,E1 156.975} C_DIS
LIN {X 0.077,Y -400.497,Z 609.656,A 0.000,B 0.000,C 90.000,E1 154.152} C_DIS
LIN {X 0.024,Y -401.161,Z 609.647,A 0.000,B 0.000,C 90.000,E1 152.410} C_DIS
LIN {X -0.148,Y -401.567,Z 609.641,A 0.000,B 0.000,C 90.000,E1 151.385} C_DIS
LIN {X -0.101,Y -402.250,Z 609.629,A 0.000,B 0.000,C 90.000,E1 149.282} C_DIS
LIN {X 0.028,Y -402.669,Z 609.622,A 0.000,B 0.000,C 90.000,E1 147.867} C_DIS
LIN {X -0.056,Y -403.186,Z 609.612,A 0.000,B 0.000,C 90.000,E1 146.135} C_DIS
LIN {X -0.127,Y -403.711,Z 609.602,A 0.000,B 0.000,C 90.000,E1 144.402} C_DIS
LIN {X 0.173,Y -404.367,Z 609.591,A 0.000,B 0.000,C 90.000,E1 142.271} C_DIS
LIN {X 0.099,Y -405.064,Z 609.579,A 0.000,B 0.000,C 90.000,E1 140.194} C_DIS
LIN {X -0.235,Y -405.466,Z 609.571,A 0.000,B 0.000,C 90.000,E1 138.852} C_DIS
LIN {X 0.108,Y -405.838,Z 609.562,A 0.000,B 0.000,C 90.000,E1 137.067} C_DIS
LIN {X -0.249,Y -406.137,Z 609.554,A 0.000,B 0.000,C 90.000,E1 135.729} C_DIS
LIN {X 0.068,Y -406.573,Z 609.540,A 0.000,B 0.000,C 90.000,E1 133.257} C_DIS
LIN {X 0.134,Y -406.878,Z 609.531,A 0.000,B 0.000,C 90.000,E1 131.515} C_DIS
LIN {X -0.177,Y -407.214,Z 609.523,A 0.000,B 0.000,C 90.000,E1 130.172} C_DIS
LIN {X 0.052,Y -407.723,Z 609.515,A 0.000,B 0.000,C 90.000,E1 128.669} C_DIS
LIN {X -0.038,Y -415.428,Z 609.500,A 0.000,B 0.000,C 90.000,E1 126.011} C_DIS
LIN {X -0.128,Y -421.038,Z 609.487,A 0.000,B 0.000,C 90.000,E1 123.706} C_DIS
LIN {X -0.167,Y -421.071,Z 609.487,A 0.000,B 0.000,C 90.000,E1 123.706} C_DIS
LIN {X 0.054,Y -423.622,Z 609.486,A 0.000,B 0.000,C 90.000,E1 123.499} C_DIS
LIN {X -0.065,Y -429.857,Z 609.484,A 0.000,B 0.000,C 90.000,E1 123.166} C_DIS
LIN {X 0.071,Y -452.370,Z 609.478,A 0.000,B 0.000,C 90.000,E1 122.005} C_DIS
LIN {X -0.033,Y -459.019,Z 609.476,A 0.000,B 0.000,C 90.000,E1 121.671} C_DIS
LIN {X -0.014,Y -467.186,Z 609.473,A 0.000,B 0.000,C 90.000,E1 121.209} C_DIS
LIN {X -0.100,Y -478.727,Z 609.470,A 0.000,B 0.000,C 90.000,E1 120.541} C_DIS
LIN {X 0.244,Y -486.827,Z 609.467,A 0.000,B 0.000,C 90.000,E1 120.001} C_DIS
LIN {X 0.115,Y -497.933,Z 609.463,A 0.000,B 0.000,C 90.000,E1 119.283} C_DIS
LIN {X -0.066,Y -504.096,Z 609.460,A 0.000,B 0.000,C 90.000,E1 118.871} C_DIS
LIN {X -0.300,Y -514.672,Z 609.456,A 0.000,B 0.000,C 90.000,E1 118.103} C_DIS
LIN {X 0.101,Y -519.132,Z 609.454,A 0.000,B 0.000,C 90.000,E1 117.719} C_DIS
LIN {X 0.280,Y -529.234,Z 609.450,A 0.000,B 0.000,C 90.000,E1 116.873} C_DIS
LIN {X 0.069,Y -536.002,Z 609.446,A 0.000,B 0.000,C 90.000,E1 116.309} C_DIS
LIN {X 0.107,Y -538.828,Z 609.445,A 0.000,B 0.000,C 90.000,E1 116.052} C_DIS
LIN {X -0.201,Y -543.951,Z 609.442,A 0.000,B 0.000,C 90.000,E1 115.591} C_DIS
LIN {X 0.141,Y -549.132,Z 609.439,A 0.000,B 0.000,C 90.000,E1 115.027} C_DIS
LIN {X -0.165,Y -553.823,Z 609.436,A 0.000,B 0.000,C 90.000,E1 114.515} C_DIS
LIN {X -0.216,Y -559.070,Z 609.432,A 0.000,B 0.000,C 90.000,E1 113.823} C_DIS
LIN {X 0.291,Y -563.528,Z 609.428,A 0.000,B 0.000,C 90.000,E1 113.078} C_DIS
LIN {X 0.107,Y -567.436,Z 609.425,A 0.000,B 0.000,C 90.000,E1 112.408} C_DIS
LIN {X 0.082,Y -571.654,Z 609.420,A 0.000,B 0.000,C 90.000,E1 111.589} C_DIS
LIN {X -0.202,Y -576.103,Z 609.415,A 0.000,B 0.000,C 90.000,E1 110.663} C_DIS
LIN {X -0.196,Y -578.486,Z 609.412,A 0.000,B 0.000,C 90.000,E1 110.120} C_DIS
LIN {X -0.135,Y -582.669,Z 609.406,A 0.000,B 0.000,C 90.000,E1 109.033} C_DIS
LIN {X -0.232,Y -585.606,Z 609.401,A 0.000,B 0.000,C 90.000,E1 108.236} C_DIS
LIN {X -0.160,Y -587.418,Z 609.398,A 0.000,B 0.000,C 90.000,E1 107.692} C_DIS
LIN {X -0.150,Y -590.638,Z 609.392,A 0.000,B 0.000,C 90.000,E1 106.622} C_DIS
LIN {X -0.088,Y -593.559,Z 609.386,A 0.000,B 0.000,C 90.000,E1 105.552} C_DIS
LIN {X -0.135,Y -600.286,Z 609.373,A 0.000,B 0.000,C 90.000,E1 103.175} C_DIS
LIN {X 0.225,Y -604.198,Z 609.366,A 0.000,B 0.000,C 90.000,E1 101.827} C_DIS
LIN {X -0.058,Y -608.080,Z 609.359,A 0.000,B 0.000,C 90.000,E1 100.546} C_DIS
LIN {X -0.274,Y -611.828,Z 609.351,A 0.000,B 0.000,C 90.000,E1 99.265} C_DIS
LIN {X 0.082,Y -615.322,Z 609.344,A 0.000,B 0.000,C 90.000,E1 97.936} C_DIS
LIN {X 0.217,Y -617.994,Z 609.338,A 0.000,B 0.000,C 90.000,E1 96.891} C_DIS
LIN {X 0.307,Y -620.520,Z 609.333,A 0.000,B 0.000,C 90.000,E1 95.853} C_DIS
LIN {X 0.127,Y -623.171,Z 609.326,A 0.000,B 0.000,C 90.000,E1 94.588} C_DIS
LIN {X -0.096,Y -624.616,Z 609.321,A 0.000,B 0.000,C 90.000,E1 93.841} C_DIS
LIN {X 0.031,Y -626.320,Z 609.316,A 0.000,B 0.000,C 90.000,E1 92.808} C_DIS
LIN {X 0.177,Y -627.820,Z 609.310,A 0.000,B 0.000,C 90.000,E1 91.776} C_DIS
LIN {X -0.302,Y -629.080,Z 609.304,A 0.000,B 0.000,C 90.000,E1 90.802} C_DIS
LIN {X 0.139,Y -629.792,Z 609.300,A 0.000,B 0.000,C 90.000,E1 90.000} C_DIS
LIN {X -0.312,Y -630.404,Z 609.294,A 0.000,B 0.000,C 90.000,E1 89.026} C_DIS
LIN {X -0.110,Y -630.588,Z 609.289,A 0.000,B 0.000,C 90.000,E1 87.993} C_DIS
LIN {X 0.070,Y -630.529,Z 609.283,A 0.000,B 0.000,C 90.000,E1 86.963} C_DIS
LIN {X -0.083,Y -630.233,Z 609.279,A 0.000,B 0.000,C 90.000,E1 86.216} C_DIS
LIN {X 0.166,Y -629.662,Z 609.273,A 0.000,B 0.000,C 90.000,E1 85.179} C_DIS
LIN {X -0.274,Y -628.809,Z 609.268,A 0.000,B 0.000,C 90.000,E1 84.204} C_DIS
LIN {X -0.041,Y -627.820,Z 609.262,A 0.000,B 0.000,C 90.000,E1 83.166} C_DIS
LIN {X 0.174,Y -626.480,Z 609.256,A 0.000,B 0.000,C 90.000,E1 82.129} C_DIS
LIN {X -0.162,Y -624.851,Z 609.251,A 0.000,B 0.000,C 90.000,E1 81.141} C_DIS
LIN {X 0.102,Y -622.932,Z 609.245,A 0.000,B 0.000,C 90.000,E1 80.095} C_DIS
LIN {X -0.273,Y -620.940,Z 609.239,A 0.000,B 0.000,C 90.000,E1 79.106} C_DIS
LIN {X 0.054,Y -618.702,Z 609.234,A 0.000,B 0.000,C 90.000,E1 78.049} C_DIS
LIN {X 0.353,Y -616.306,Z 609.228,A 0.000,B 0.000,C 90.000,E1 76.992} C_DIS
LIN {X -0.221,Y -613.051,Z 609.221,A 0.000,B 0.000,C 90.000,E1 75.755} C_DIS
LIN {X -0.014,Y -610.262,Z 609.215,A 0.000,B 0.000,C 90.000,E1 74.700} C_DIS
LIN {X -0.021,Y -608.005,Z 609.211,A 0.000,B 0.000,C 90.000,E1 73.921} C_DIS
LIN {X -0.047,Y -605.623,Z 609.206,A 0.000,B 0.000,C 90.000,E1 73.142} C_DIS
LIN {X 0.176,Y -603.983,Z 609.203,A 0.000,B 0.000,C 90.000,E1 72.598} C_DIS
LIN {X 0.202,Y -602.177,Z 609.201,A 0.000,B 0.000,C 90.000,E1 72.072} C_DIS
LIN {X 0.301,Y -599.134,Z 609.196,A 0.000,B 0.000,C 90.000,E1 71.275} C_DIS
LIN {X 0.178,Y -595.841,Z 609.192,A 0.000,B 0.000,C 90.000,E1 70.496} C_DIS
LIN {X 0.220,Y -592.352,Z 609.187,A 0.000,B 0.000,C 90.000,E1 69.699} C_DIS
LIN {X 0.227,Y -588.686,Z 609.183,A 0.000,B 0.000,C 90.000,E1 68.901} C_DIS
LIN {X 0.125,Y -583.908,Z 609.178,A 0.000,B 0.000,C 90.000,E1 67.975} C_DIS
LIN {X -0.361,Y -581.083,Z 609.175,A 0.000,B 0.000,C 90.000,E1 67.486} C_DIS
LIN {X -0.252,Y -576.234,Z 609.170,A 0.000,B 0.000,C 90.000,E1 66.666} C_DIS
LIN {X 0.208,Y -572.967,Z 609.167,A 0.000,B 0.000,C 90.000,E1 66.102} C_DIS
LIN {X 0.084,Y -568.280,Z 609.164,A 0.000,B 0.000,C 90.000,E1 65.433} C_DIS
LIN {X -0.272,Y -564.084,Z 609.161,A 0.000,B 0.000,C 90.000,E1 64.921} C_DIS
LIN {X 0.098,Y -559.613,Z 609.158,A 0.000,B 0.000,C 90.000,E1 64.332} C_DIS
LIN {X -0.166,Y -555.934,Z 609.155,A 0.000,B 0.000,C 90.000,E1 63.948} C_DIS
LIN {X 0.267,Y -554.808,Z 609.154,A 0.000,B 0.000,C 90.000,E1 63.768} C_DIS
LIN {X -0.093,Y -549.876,Z 609.152,A 0.000,B 0.000,C 90.000,E1 63.307} C_DIS
LIN {X -0.084,Y -544.514,Z 609.149,A 0.000,B 0.000,C 90.000,E1 62.820} C_DIS
LIN {X 0.080,Y -538.915,Z 609.147,A 0.000,B 0.000,C 90.000,E1 62.359} C_DIS
LIN {X -0.024,Y -533.802,Z 609.145,A 0.000,B 0.000,C 90.000,E1 62.025} C_DIS
LIN {X -0.197,Y -527.217,Z 609.142,A 0.000,B 0.000,C 90.000,E1 61.641} C_DIS
LIN {X -0.089,Y -520.468,Z 609.140,A 0.000,B 0.000,C 90.000,E1 61.257} C_DIS
LIN {X 0.053,Y -515.379,Z 609.139,A 0.000,B 0.000,C 90.000,E1 60.973} C_DIS
LIN {X -0.074,Y -503.298,Z 609.136,A 0.000,B 0.000,C 90.000,E1 60.411} C_DIS
LIN {X -0.101,Y -486.253,Z 609.131,A 0.000,B 0.000,C 90.000,E1 59.616} C_DIS
LIN {X -0.259,Y -474.524,Z 609.128,A 0.000,B 0.000,C 90.000,E1 59.076} C_DIS
LIN {X -0.105,Y -464.679,Z 609.125,A 0.000,B 0.000,C 90.000,E1 58.584} C_DIS
LIN {X 0.144,Y -445.944,Z 609.120,A 0.000,B 0.000,C 90.000,E1 57.582} C_DIS
LIN {X 0.103,Y -445.932,Z 609.120,A 0.000,B 0.000,C 90.000,E1 57.582} C_DIS
LIN {X 0.051,Y -444.056,Z 609.114,A 0.000,B 0.000,C 90.000,E1 56.548} C_DIS
LIN {X 0.095,Y -434.253,Z 609.091,A 0.000,B 0.000,C 90.000,E1 52.271} C_DIS
LIN {X -0.062,Y -431.764,Z 609.083,A 0.000,B 0.000,C 90.000,E1 50.964} C_DIS
LIN {X 0.118,Y -430.181,Z 609.079,A 0.000,B 0.000,C 90.000,E1 50.275} C_DIS
LIN {X 0.116,Y -429.875,Z 609.079,A 0.000,B 0.000,C 90.000,E1 50.150} C_DIS
LIN {X 0.101,Y -430.861,Z 609.070,A 0.000,B 0.000,C 90.000,E1 48.609} C_DIS
LIN {X -0.156,Y -431.612,Z 609.063,A 0.000,B 0.000,C 90.000,E1 47.310} C_DIS
LIN {X 0.002,Y -432.837,Z 609.050,A 0.000,B 0.000,C 90.000,E1 44.960} C_DIS
LIN {X -0.061,Y -434.054,Z 609.039,A 0.000,B 0.000,C 90.000,E1 42.975} C_DIS
LIN {X -0.008,Y -434.938,Z 609.030,A 0.000,B 0.000,C 90.000,E1 41.310} C_DIS
LIN {X -0.205,Y -435.604,Z 609.022,A 0.000,B 0.000,C 90.000,E1 40.011} C_DIS
LIN {X -0.058,Y -436.378,Z 609.013,A 0.000,B 0.000,C 90.000,E1 38.338} C_DIS
LIN {X 0.093,Y -436.903,Z 609.006,A 0.000,B 0.000,C 90.000,E1 36.996} C_DIS
LIN {X 0.018,Y -437.464,Z 608.995,A 0.000,B 0.000,C 90.000,E1 35.025} C_DIS
LIN {X 0.013,Y -437.807,Z 608.987,A 0.000,B 0.000,C 90.000,E1 33.706} C_DIS
LIN {X -0.227,Y -438.037,Z 608.980,A 0.000,B 0.000,C 90.000,E1 32.418} C_DIS
LIN {X -0.015,Y -438.476,Z 608.969,A 0.000,B 0.000,C 90.000,E1 30.413} C_DIS
LIN {X 0.023,Y -438.956,Z 608.956,A 0.000,B 0.000,C 90.000,E1 28.103} C_DIS
LIN {X -0.214,Y -439.336,Z 608.947,A 0.000,B 0.000,C 90.000,E1 26.488} C_DIS
LIN {X -0.058,Y -439.759,Z 608.938,A 0.000,B 0.000,C 90.000,E1 24.823} C_DIS
LIN {X 0.161,Y -440.326,Z 608.927,A 0.000,B 0.000,C 90.000,E1 22.823} C_DIS
LIN {X -0.194,Y -440.860,Z 608.918,A 0.000,B 0.000,C 90.000,E1 21.227} C_DIS
LIN {X -0.122,Y -441.485,Z 608.909,A 0.000,B 0.000,C 90.000,E1 19.577} C_DIS
LIN {X -0.068,Y -442.376,Z 608.896,A 0.000,B 0.000,C 90.000,E1 17.275} C_DIS
LIN {X 0.171,Y -443.407,Z 608.883,A 0.000,B 0.000,C 90.000,E1 14.954} C_DIS
LIN {X 0.057,Y -444.887,Z 608.869,A 0.000,B 0.000,C 90.000,E1 12.355} C_DIS
LIN {X 0.226,Y -446.695,Z 608.854,A 0.000,B 0.000,C 90.000,E1 9.726} C_DIS
LIN {X 0.052,Y -448.444,Z 608.842,A 0.000,B 0.000,C 90.000,E1 7.473} C_DIS
LIN {X -0.070,Y -450.449,Z 608.829,A 0.000,B 0.000,C 90.000,E1 5.220} C_DIS
LIN {X 0.029,Y -452.423,Z 608.818,A 0.000,B 0.000,C 90.000,E1 3.269} C_DIS
LIN {X -0.103,Y -454.952,Z 608.806,A 0.000,B 0.000,C 90.000,E1 1.031} C_DIS
LIN {X 0.195,Y -458.672,Z 608.790,A 0.000,B 0.000,C 90.000,E1 358.167} C_DIS
LIN {X 0.202,Y -462.957,Z 608.774,A 0.000,B 0.000,C 90.000,E1 355.298} C_DIS
LIN {X 0.225,Y -466.071,Z 608.763,A 0.000,B 0.000,C 90.000,E1 353.394} C_DIS
LIN {X 0.051,Y -468.634,Z 608.755,A 0.000,B 0.000,C 90.000,E1 351.837} C_DIS
LIN {X -0.197,Y -471.610,Z 608.744,A 0.000,B 0.000,C 90.000,E1 349.982} C_DIS
LIN {X -0.230,Y -476.326,Z 608.729,A 0.000,B 0.000,C 90.000,E1 347.173} C_DIS
LIN {X 0.273,Y -480.802,Z 608.715,A 0.000,B 0.000,C 90.000,E1 344.629} C_DIS
LIN {X 0.112,Y -484.811,Z 608.703,A 0.000,B 0.000,C 90.000,E1 342.489} C_DIS
LIN {X 0.003,Y -487.752,Z 608.694,A 0.000,B 0.000,C 90.000,E1 340.967} C_DIS
LIN {X -0.043,Y -490.685,Z 608.686,A 0.000,B 0.000,C 90.000,E1 339.444} C_DIS
LIN {X -0.042,Y -493.584,Z 608.677,A 0.000,B 0.000,C 90.000,E1 337.922} C_DIS
LIN {X -0.125,Y -495.644,Z 608.671,A 0.000,B 0.000,C 90.000,E1 336.719} C_DIS
LIN {X 0.140,Y -498.113,Z 608.662,A 0.000,B 0.000,C 90.000,E1 335.177} C_DIS
LIN {X -0.038,Y -500.443,Z 608.654,A 0.000,B 0.000,C 90.000,E1 333.691} C_DIS
LIN {X -0.010,Y -502.190,Z 608.647,A 0.000,B 0.000,C 90.000,E1 332.487} C_DIS
LIN {X -0.110,Y -504.422,Z 608.639,A 0.000,B 0.000,C 90.000,E1 331.001} C_DIS
LIN {X -0.048,Y -507.043,Z 608.629,A 0.000,B 0.000,C 90.000,E1 329.203} C_DIS
LIN {X -0.071,Y -514.364,Z 608.606,A 0.000,B 0.000,C 90.000,E1 325.055} C_DIS
LIN {X -0.141,Y -518.761,Z 608.594,A 0.000,B 0.000,C 90.000,E1 323.004} C_DIS
LIN {X 0.002,Y -520.854,Z 608.590,A 0.000,B 0.000,C 90.000,E1 322.110} C_DIS
LIN {X -0.072,Y -522.520,Z 608.586,A 0.000,B 0.000,C 90.000,E1 321.537} C_DIS
LIN {X 0.157,Y -523.327,Z 608.585,A 0.000,B 0.000,C 90.000,E1 321.331} C_DIS
LIN {X 0.254,Y -524.900,Z 608.583,A 0.000,B 0.000,C 90.000,E1 320.884} C_DIS
LIN {X -0.340,Y -525.580,Z 608.582,A 0.000,B 0.000,C 90.000,E1 320.803} C_DIS
LIN {X 0.166,Y -527.702,Z 608.580,A 0.000,B 0.000,C 90.000,E1 320.436} C_DIS
LIN {X 0.189,Y -531.390,Z 608.578,A 0.000,B 0.000,C 90.000,E1 319.989} C_DIS
LIN {X 0.136,Y -536.881,Z 608.575,A 0.000,B 0.000,C 90.000,E1 319.461} C_DIS
LIN {X 0.053,Y -544.046,Z 608.571,A 0.000,B 0.000,C 90.000,E1 318.852} C_DIS
LIN {X -0.133,Y -549.712,Z 608.569,A 0.000,B 0.000,C 90.000,E1 318.447} C_DIS
LIN {X 0.025,Y -561.317,Z 608.564,A 0.000,B 0.000,C 90.000,E1 317.514} C_DIS
LIN {X 0.164,Y -583.265,Z 608.555,A 0.000,B 0.000,C 90.000,E1 315.810} C_DIS
LIN {X -0.245,Y -588.971,Z 608.552,A 0.000,B 0.000,C 90.000,E1 315.405} C_DIS
LIN {X 0.056,Y -594.445,Z 608.550,A 0.000,B 0.000,C 90.000,E1 314.919} C_DIS
LIN {X -0.349,Y -602.561,Z 608.546,A 0.000,B 0.000,C 90.000,E1 314.271} C_DIS
LIN {X 0.121,Y -608.941,Z 608.542,A 0.000,B 0.000,C 90.000,E1 313.623} C_DIS
LIN {X 0.041,Y -612.677,Z 608.540,A 0.000,B 0.000,C 90.000,E1 313.257} C_DIS
LIN {X 0.059,Y -619.827,Z 608.536,A 0.000,B 0.000,C 90.000,E1 312.486} C_DIS
LIN {X -0.012,Y -627.545,Z 608.531,A 0.000,B 0.000,C 90.000,E1 311.595} C_DIS
LIN {X 0.443,Y -635.833,Z 608.526,A 0.000,B 0.000,C 90.000,E1 310.539} C_DIS
LIN {X -0.290,Y -642.790,Z 608.521,A 0.000,B 0.000,C 90.000,E1 309.725} C_DIS
LIN {X -0.053,Y -648.329,Z 608.516,A 0.000,B 0.000,C 90.000,E1 308.955} C_DIS
LIN {X -0.086,Y -652.586,Z 608.513,A 0.000,B 0.000,C 90.000,E1 308.338} C_DIS
LIN {X -0.159,Y -657.156,Z 608.509,A 0.000,B 0.000,C 90.000,E1 307.604} C_DIS
LIN {X 0.296,Y -660.630,Z 608.505,A 0.000,B 0.000,C 90.000,E1 306.950} C_DIS
LIN {X -0.150,Y -663.796,Z 608.502,A 0.000,B 0.000,C 90.000,E1 306.377} C_DIS
LIN {X -0.088,Y -666.170,Z 608.499,A 0.000,B 0.000,C 90.000,E1 305.884} C_DIS
LIN {X -0.013,Y -668.342,Z 608.497,A 0.000,B 0.000,C 90.000,E1 305.391} C_DIS
LIN {X 0.041,Y -671.338,Z 608.493,A 0.000,B 0.000,C 90.000,E1 304.659} C_DIS
LIN {X 0.042,Y -675.922,Z 608.486,A 0.000,B 0.000,C 90.000,E1 303.452} C_DIS
LIN {X -0.075,Y -680.111,Z 608.479,A 0.000,B 0.000,C 90.000,E1 302.260} C_DIS
LIN {X 0.281,Y -684.956,Z 608.471,A 0.000,B 0.000,C 90.000,E1 300.797} C_DIS
LIN {X -0.200,Y -689.622,Z 608.463,A 0.000,B 0.000,C 90.000,E1 299.411} C_DIS
LIN {X 0.133,Y -692.626,Z 608.458,A 0.000,B 0.000,C 90.000,E1 298.437} C_DIS
LIN {X 0.144,Y -696.000,Z 608.452,A 0.000,B 0.000,C 90.000,E1 297.257} C_DIS
LIN {X -0.019,Y -697.758,Z 608.448,A 0.000,B 0.000,C 90.000,E1 296.565} C_DIS
LIN {X 0.147,Y -698.563,Z 608.444,A 0.000,B 0.000,C 90.000,E1 295.848} C_DIS
LIN {X 0.011,Y -697.410,Z 608.440,A 0.000,B 0.000,C 90.000,E1 295.155} C_DIS
LIN {X 0.142,Y -696.926,Z 608.439,A 0.000,B 0.000,C 90.000,E1 295.027} C_DIS
LIN {X -0.137,Y -692.815,Z 608.436,A 0.000,B 0.000,C 90.000,E1 294.463} C_DIS
LIN {X -0.013,Y -691.497,Z 608.435,A 0.000,B 0.000,C 90.000,E1 294.335} C_DIS
LIN {X -0.004,Y -687.671,Z 608.434,A 0.000,B 0.000,C 90.000,E1 294.131} C_DIS
LIN {X 0.197,Y -684.183,Z 608.433,A 0.000,B 0.000,C 90.000,E1 293.951} C_DIS
LIN {X -0.112,Y -682.363,Z 608.433,A 0.000,B 0.000,C 90.000,E1 293.898} C_DIS
LIN {X 0.067,Y -675.425,Z 608.432,A 0.000,B 0.000,C 90.000,E1 293.695} C_DIS
LIN {X -0.132,Y -661.812,Z 608.431,A 0.000,B 0.000,C 90.000,E1 293.515} C_DIS
LIN {X -0.303,Y -647.721,Z 608.430,A 0.000,B 0.000,C 90.000,E1 293.334} C_DIS
LIN {X -0.181,Y -634.513,Z 608.428,A 0.000,B 0.000,C 90.000,E1 293.078} C_DIS
LIN {X 0.164,Y -624.639,Z 608.427,A 0.000,B 0.000,C 90.000,E1 292.823} C_DIS
LIN {X -0.214,Y -608.172,Z 608.424,A 0.000,B 0.000,C 90.000,E1 292.386} C_DIS
LIN {X 0.161,Y -583.976,Z 608.420,A 0.000,B 0.000,C 90.000,E1 291.589} C_DIS
LIN {X -0.241,Y -576.715,Z 608.419,A 0.000,B 0.000,C 90.000,E1 291.408} C_DIS
LIN {X -0.154,Y -566.626,Z 608.417,A 0.000,B 0.000,C 90.000,E1 291.099} C_DIS
LIN {X -0.166,Y -565.050,Z 608.417,A 0.000,B 0.000,C 90.000,E1 291.046} C_DIS
LIN {X -0.023,Y -560.111,Z 608.416,A 0.000,B 0.000,C 90.000,E1 290.791} C_DIS
LIN {X -0.073,Y -560.015,Z 608.416,A 0.000,B 0.000,C 90.000,E1 290.791} C_DIS
LIN {X -0.184,Y -558.353,Z 608.414,A 0.000,B 0.000,C 90.000,E1 290.610} C_DIS
LIN {X -0.226,Y -558.339,Z 608.414,A 0.000,B 0.000,C 90.000,E1 290.610} C_DIS
LIN {X -0.006,Y -557.876,Z 608.413,A 0.000,B 0.000,C 90.000,E1 290.375} C_DIS
LIN {X 0.069,Y -557.608,Z 608.410,A 0.000,B 0.000,C 90.000,E1 289.812} C_DIS
LIN {X 0.127,Y -557.703,Z 608.402,A 0.000,B 0.000,C 90.000,E1 288.417} C_DIS
LIN {X -0.112,Y -557.531,Z 608.396,A 0.000,B 0.000,C 90.000,E1 287.330} C_DIS
LIN {X 0.301,Y -557.105,Z 608.389,A 0.000,B 0.000,C 90.000,E1 285.898} C_DIS
LIN {X 0.156,Y -556.739,Z 608.384,A 0.000,B 0.000,C 90.000,E1 285.079} C_DIS
LIN {X 0.143,Y -555.911,Z 608.375,A 0.000,B 0.000,C 90.000,E1 283.411} C_DIS
LIN {X 0.259,Y -555.204,Z 608.367,A 0.000,B 0.000,C 90.000,E1 282.007} C_DIS
LIN {X 0.101,Y -554.033,Z 608.354,A 0.000,B 0.000,C 90.000,E1 279.792} C_DIS
LIN {X -0.224,Y -553.027,Z 608.344,A 0.000,B 0.000,C 90.000,E1 277.871} C_DIS
LIN {X -0.138,Y -552.025,Z 608.331,A 0.000,B 0.000,C 90.000,E1 275.625} C_DIS
LIN {X -0.230,Y -551.425,Z 608.322,A 0.000,B 0.000,C 90.000,E1 273.955} C_DIS
LIN {X 0.140,Y -550.927,Z 608.313,A 0.000,B 0.000,C 90.000,E1 272.236} C_DIS
LIN {X -0.103,Y -550.577,Z 608.305,A 0.000,B 0.000,C 90.000,E1 270.859} C_DIS
LIN {X 0.186,Y -550.135,Z 608.297,A 0.000,B 0.000,C 90.000,E1 269.427} C_DIS
LIN {X -0.143,Y -549.711,Z 608.291,A 0.000,B 0.000,C 90.000,E1 268.339} C_DIS
LIN {X 0.136,Y -549.150,Z 608.283,A 0.000,B 0.000,C 90.000,E1 266.906} C_DIS
LIN {X -0.110,Y -548.519,Z 608.275,A 0.000,B 0.000,C 90.000,E1 265.527} C_DIS
LIN {X 0.147,Y -547.868,Z 608.269,A 0.000,B 0.000,C 90.000,E1 264.375} C_DIS
LIN {X -0.150,Y -547.170,Z 608.263,A 0.000,B 0.000,C 90.000,E1 263.280} C_DIS
LIN {X 0.081,Y -546.240,Z 608.256,A 0.000,B 0.000,C 90.000,E1 262.129} C_DIS
LIN {X 0.009,Y -544.652,Z 608.247,A 0.000,B 0.000,C 90.000,E1 260.443} C_DIS
LIN {X 0.074,Y -542.475,Z 608.234,A 0.000,B 0.000,C 90.000,E1 258.173} C_DIS
LIN {X 0.144,Y -540.871,Z 608.225,A 0.000,B 0.000,C 90.000,E1 256.464} C_DIS
LIN {X 0.045,Y -539.791,Z 608.219,A 0.000,B 0.000,C 90.000,E1 255.338} C_DIS
LIN {X 0.199,Y -538.013,Z 608.209,A 0.000,B 0.000,C 90.000,E1 253.614} C_DIS
LIN {X -0.003,Y -535.985,Z 608.198,A 0.000,B 0.000,C 90.000,E1 251.638} C_DIS
LIN {X -0.031,Y -534.703,Z 608.192,A 0.000,B 0.000,C 90.000,E1 250.496} C_DIS
LIN {X 0.080,Y -533.525,Z 608.187,A 0.000,B 0.000,C 90.000,E1 249.625} C_DIS
LIN {X 0.196,Y -531.695,Z 608.181,A 0.000,B 0.000,C 90.000,E1 248.465} C_DIS
LIN {X -0.028,Y -529.187,Z 608.173,A 0.000,B 0.000,C 90.000,E1 247.050} C_DIS
LIN {X -0.096,Y -526.477,Z 608.164,A 0.000,B 0.000,C 90.000,E1 245.613} C_DIS
LIN {X -0.155,Y -524.062,Z 608.158,A 0.000,B 0.000,C 90.000,E1 244.460} C_DIS
LIN {X 0.225,Y -521.592,Z 608.152,A 0.000,B 0.000,C 90.000,E1 243.256} C_DIS
LIN {X 0.095,Y -518.955,Z 608.145,A 0.000,B 0.000,C 90.000,E1 242.103} C_DIS
LIN {X 0.169,Y -516.197,Z 608.139,A 0.000,B 0.000,C 90.000,E1 240.923} C_DIS
LIN {X 0.106,Y -511.293,Z 608.127,A 0.000,B 0.000,C 90.000,E1 238.869} C_DIS
LIN {X -0.105,Y -508.410,Z 608.121,A 0.000,B 0.000,C 90.000,E1 237.709} C_DIS
LIN {X 0.068,Y -505.243,Z 608.114,A 0.000,B 0.000,C 90.000,E1 236.501} C_DIS
LIN {X -0.063,Y -501.130,Z 608.106,A 0.000,B 0.000,C 90.000,E1 235.022} C_DIS
LIN {X -0.128,Y -495.394,Z 608.094,A 0.000,B 0.000,C 90.000,E1 232.924} C_DIS
LIN {X 0.160,Y -491.542,Z 608.086,A 0.000,B 0.000,C 90.000,E1 231.376} C_DIS
LIN {X 0.061,Y -487.598,Z 608.077,A 0.000,B 0.000,C 90.000,E1 229.865} C_DIS
LIN {X 0.139,Y -483.755,Z 608.069,A 0.000,B 0.000,C 90.000,E1 228.324} C_DIS
LIN {X -0.077,Y -479.146,Z 608.058,A 0.000,B 0.000,C 90.000,E1 226.500} C_DIS
LIN {X -0.054,Y -474.585,Z 608.048,A 0.000,B 0.000,C 90.000,E1 224.636} C_DIS
LIN {X 0.101,Y -471.010,Z 608.039,A 0.000,B 0.000,C 90.000,E1 223.056} C_DIS
LIN {X -0.128,Y -467.462,Z 608.031,A 0.000,B 0.000,C 90.000,E1 221.515} C_DIS
LIN {X -0.162,Y -461.987,Z 608.017,A 0.000,B 0.000,C 90.000,E1 218.991} C_DIS
LIN {X -0.117,Y -458.046,Z 608.006,A 0.000,B 0.000,C 90.000,E1 217.076} C_DIS
LIN {X -0.086,Y -454.274,Z 607.995,A 0.000,B 0.000,C 90.000,E1 215.152} C_DIS
SetRPM(0)
End
